KUKA KRL program: EPS_2_251455_MH56A_A_20251003061556.src

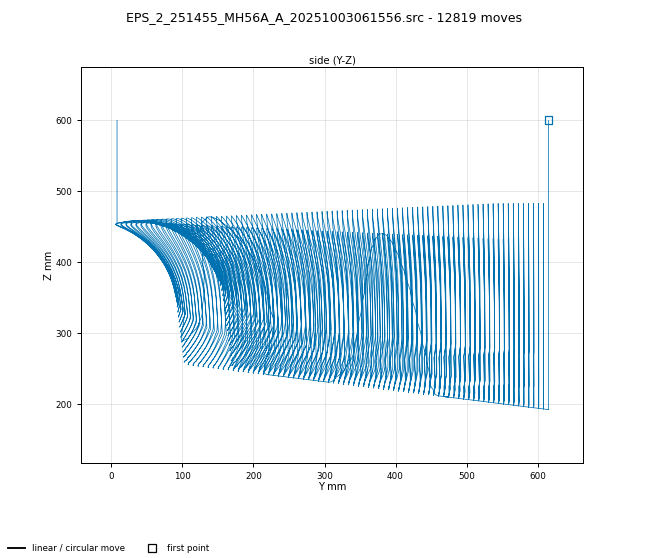
[picture p0: tool path of EPS_2_251455_MH56A_A_20251003061556.src, 12819 of 12821 moves have a stored position in this frame; points joined in program order, loops and branches not executed]
&ACCESS RVP
&REL 4
&COMMENT QRS 19112012
&PARAM EDITMASK = *
DEF PART()
EXT BAS (BAS_COMMAND :IN,REAL :IN )
INT I
BAS (#INITMOV,0 )

;KUKA QRS Post kuka4.cps  Date:22-06-2017 !

File_ID=2879

QRS_PRE_INIT()

;Init var - Until changes are made in qrs_pre_init
Outlet_Square_prg=0
Inlet_1_Square_prg=0
Inlet_2_Square_prg=0
Inlet_3_Square_prg=0
Inlet_4_Square_prg=0
Inlet_5_Square_prg=0

Outlet_1={X 0.000, Y 540.910, Z 382.500, B 0.000, E1 0.000 }
Inlet_1={X 0.000, Y 544.470, Z 332.500, B 0.000, E1 191.000 }
Outlet_1_type=201
Inlet_1_type=201
;QRS#1=Sidecore dimensions
;QRS#2=200-8" PVC SDR 35
;QRS#3=200-8" PVC SDR 35
;QRS#4=
;QRS#5=
;QRS#6=
;QRS#7=
;QRS#8=
;QRS#9=12-08 PSX
;QRS#10=12-08 PSX
;QRS#11=
;QRS#12=
;QRS#13=
;QRS#14=
;QRS#15=
;QRS#16=1220x127x762 2,5'
;QRS#17=EPS Height
;QRS#18=483
;QRS#19=*
;QRS#20= UPDATED VERSION 22-06-2017
;QRS#21=*
Outlet_Square=0100
Inlet_1_Square=0100
Inlet_2_Square=0
Inlet_3_Square=0
Inlet_4_Square=0
Inlet_5_Square=0
Mill_Square=1
Outlet_Square_Prg=204
Inlet_1_Square_prg=204

QRS_INIT()

$ADVANCE=5

; T1
PTP {E1 173.577,E2 173.577}
PTP {X 0,Y 615.465,A -85,B 0,C 180,E1 173.577,E2 173.577,E3 0,E4 0,E5 0,E6 0}
QRS_SPEED_INIT()
LIN {X 0,Y 615.465,Z 600,A -85,B 0,C 180,E1 173.577,E2 173.577,E3 0,E4 0,E5 0,E6 0} C_VEL
LIN {X 0,Y 615.465,Z 202.872,A -85,B 0,C 180,E1 173.577,E2 173.577} C_VEL
LIN {X 0,Y 615.465,Z 194.7,A -85,B 0,C 180,E1 173.577,E2 173.577} C_VEL
LIN {X 0,Y 615.452,Z 192.7,A -85,B 0,C 180,E1 173.391,E2 173.391} C_VEL
LIN {X 0,Y 615.455,Z 192.7,A -85,B 0,C 180,E1 170.801,E2 170.801} C_VEL
LIN {X 0,Y 615.413,Z 192.699,A -85,B 0,C 180,E1 168.138,E2 168.138} C_VEL
LIN {X 0,Y 615.463,Z 192.7,A -85,B 0,C 180,E1 165.45,E2 165.45} C_VEL
LIN {X 0,Y 615.439,Z 192.698,A -85,B 0,C 180,E1 162.728,E2 162.728} C_VEL
LIN {X 0,Y 615.432,Z 192.698,A -85,B 0,C 180,E1 160.66,E2 160.66} C_VEL
LIN {X 0,Y 615.425,Z 192.698,A -85,B 0,C 180,E1 158.566,E2 158.566} C_VEL
LIN {X 0,Y 615.42,Z 192.698,A -85,B 0,C 180,E1 156.441,E2 156.441} C_VEL
LIN {X 0,Y 615.42,Z 192.698,A -85,B 0,C 180,E1 154.281,E2 154.281} C_VEL
LIN {X 0,Y 615.482,Z 192.701,A -85,B 0,C 180,E1 151.538,E2 151.538} C_VEL
LIN {X 0,Y 615.445,Z 192.696,A -85,B 0,C 180,E1 148.909,E2 148.909} C_VEL
LIN {X 0,Y 615.423,Z 192.697,A -85,B 0,C 180,E1 146.464,E2 146.464} C_VEL
LIN {X 0,Y 615.435,Z 192.698,A -85,B 0,C 180,E1 144.163,E2 144.163} C_VEL
LIN {X 0,Y 615.459,Z 192.699,A -85,B 0,C 180,E1 141.929,E2 141.929} C_VEL
LIN {X 0,Y 615.488,Z 192.693,A -85,B 0,C 180,E1 139.393,E2 139.393} C_VEL
LIN {X 0,Y 615.431,Z 192.695,A -85,B 0,C 180,E1 136.75,E2 136.75} C_VEL
LIN {X 0,Y 615.467,Z 192.699,A -85,B 0,C 180,E1 133.995,E2 133.995} C_VEL
LIN {X 0,Y 615.448,Z 192.693,A -85,B 0,C 180,E1 131.09,E2 131.09} C_VEL
LIN {X 0,Y 615.434,Z 192.695,A -85,B 0,C 180,E1 128.902,E2 128.902} C_VEL
LIN {X 0,Y 615.444,Z 192.697,A -85,B 0,C 180,E1 126.422,E2 126.422} C_VEL
LIN {X 0,Y 615.485,Z 192.69,A -85,B 0,C 180,E1 123.533,E2 123.533} C_VEL
LIN {X 0,Y 615.438,Z 192.694,A -85,B 0,C 180,E1 120.918,E2 120.918} C_VEL
LIN {X 0,Y 615.454,Z 192.697,A -85,B 0,C 180,E1 118.444,E2 118.444} C_VEL
LIN {X 0,Y 615.48,Z 192.689,A -85,B 0,C 180,E1 115.566,E2 115.566} C_VEL
LIN {X 0,Y 615.476,Z 192.689,A -85,B 0,C 180,E1 113.553,E2 113.553} C_VEL
LIN {X 0,Y 615.459,Z 192.69,A -85,B 0,C 180,E1 111.429,E2 111.429} C_VEL
LIN {X 0,Y 615.454,Z 192.691,A -85,B 0,C 180,E1 109.336,E2 109.336} C_VEL
LIN {X 0,Y 615.449,Z 192.691,A -85,B 0,C 180,E1 107.269,E2 107.269} C_VEL
LIN {X 0,Y 615.448,Z 192.692,A -85,B 0,C 180,E1 105.224,E2 105.224} C_VEL
LIN {X 0,Y 615.445,Z 192.692,A -85,B 0,C 180,E1 103.2,E2 103.2} C_VEL
LIN {X 0,Y 615.479,Z 192.698,A -85,B 0,C 180,E1 100.525,E2 100.525} C_VEL
LIN {X 0,Y 615.485,Z 192.688,A -85,B 0,C 180,E1 97.874,E2 97.874} C_VEL
LIN {X 0,Y 615.452,Z 192.79,A -85,B 0,C 180,E1 96.973,E2 96.973} C_VEL
LIN {X 0,Y 615.487,Z 208.3,A -85,B 0,C 180,E1 94.255,E2 94.255} C_VEL
LIN {X 0,Y 615.493,Z 222.362,A -85,B 0,C 180,E1 91.818,E2 91.818} C_VEL
LIN {X 0,Y 615.459,Z 329.633,A -85,B 0,C 180,E1 90.53,E2 90.53} C_VEL
LIN {X 0,Y 615.475,Z 342.412,A -85,B 0,C 180,E1 90.244,E2 90.244} C_VEL
LIN {X 0,Y 615.497,Z 354.793,A -85,B 0,C 180,E1 89.835,E2 89.835} C_VEL
LIN {X 0,Y 615.468,Z 365.91,A -85,B 0,C 180,E1 89.345,E2 89.345} C_VEL
LIN {X 0,Y 615.467,Z 377.404,A -85,B 0,C 180,E1 88.69,E2 88.69} C_VEL
LIN {X 0,Y 615.498,Z 388.761,A -85,B 0,C 180,E1 87.872,E2 87.872} C_VEL
LIN {X 0,Y 615.498,Z 397.906,A -85,B 0,C 180,E1 87.054,E2 87.054} C_VEL
LIN {X 0,Y 615.496,Z 406.784,A -85,B 0,C 180,E1 86.071,E2 86.071} C_VEL
LIN {X 0,Y 615.496,Z 413.964,A -85,B 0,C 180,E1 85.087,E2 85.087} C_VEL
LIN {X 0,Y 615.499,Z 419.723,A -85,B 0,C 180,E1 84.101,E2 84.101} C_VEL
LIN {X 0,Y 615.495,Z 424.321,A -85,B 0,C 180,E1 83.101,E2 83.101} C_VEL
LIN {X 0,Y 615.497,Z 427.731,A -85,B 0,C 180,E1 82.124,E2 82.124} C_VEL
LIN {X 0,Y 615.495,Z 429.484,A -85,B 0,C 180,E1 81.463,E2 81.463} C_VEL
LIN {X 0,Y 615.499,Z 431.728,A -85,B 0,C 180,E1 80.138,E2 80.138} C_VEL
LIN {X 0,Y 615.495,Z 432.357,A -85,B 0,C 180,E1 79.11,E2 79.11} C_VEL
LIN {X 0,Y 615.494,Z 432.06,A -85,B 0,C 180,E1 78.139,E2 78.139} C_VEL
LIN {X 0,Y 615.496,Z 431.373,A -85,B 0,C 180,E1 77.47,E2 77.47} C_VEL
LIN {X 0,Y 615.496,Z 430.246,A -85,B 0,C 180,E1 76.799,E2 76.799} C_VEL
LIN {X 0,Y 615.499,Z 428.503,A -85,B 0,C 180,E1 76.065,E2 76.065} C_VEL
LIN {X 0,Y 615.497,Z 425.464,A -85,B 0,C 180,E1 75.113,E2 75.113} C_VEL
LIN {X 0,Y 615.496,Z 421.132,A -85,B 0,C 180,E1 74.095,E2 74.095} C_VEL
LIN {X 0,Y 615.498,Z 415.52,A -85,B 0,C 180,E1 73.072,E2 73.072} C_VEL
LIN {X 0,Y 615.499,Z 408.424,A -85,B 0,C 180,E1 72.044,E2 72.044} C_VEL
LIN {X 0,Y 615.497,Z 401.088,A -85,B 0,C 180,E1 71.182,E2 71.182} C_VEL
LIN {X 0,Y 615.498,Z 391.05,A -85,B 0,C 180,E1 70.229,E2 70.229} C_VEL
LIN {X 0,Y 615.489,Z 380.813,A -85,B 0,C 180,E1 69.444,E2 69.444} C_VEL
LIN {X 0,Y 615.462,Z 369.296,A -85,B 0,C 180,E1 68.744,E2 68.744} C_VEL
LIN {X 0,Y 615.491,Z 357.249,A -85,B 0,C 180,E1 68.173,E2 68.173} C_VEL
LIN {X 0,Y 615.446,Z 345.875,A -85,B 0,C 180,E1 67.764,E2 67.764} C_VEL
LIN {X 0,Y 615.433,Z 333.072,A -85,B 0,C 180,E1 67.442,E2 67.442} C_VEL
LIN {X 0,Y 615.436,Z 317.595,A -85,B 0,C 180,E1 67.218,E2 67.218} C_VEL
LIN {X 0,Y 615.479,Z 222.383,A -85,B 0,C 180,E1 66.095,E2 66.095} C_VEL
LIN {X 0,Y 615.491,Z 206.009,A -85,B 0,C 180,E1 63.257,E2 63.257} C_VEL
LIN {X 0,Y 615.469,Z 192.69,A -85,B 0,C 180,E1 60.899,E2 60.899} C_VEL
LIN {X 0,Y 615.489,Z 192.684,A -85,B 0,C 180,E1 58.317,E2 58.317} C_VEL
LIN {X 0,Y 615.483,Z 192.692,A -85,B 0,C 180,E1 55.98,E2 55.98} C_VEL
LIN {X 0,Y 615.484,Z 192.701,A -85,B 0,C 180,E1 53.578,E2 53.578} C_VEL
LIN {X 0,Y 615.462,Z 192.689,A -85,B 0,C 180,E1 50.941,E2 50.941} C_VEL
LIN {X 0,Y 615.489,Z 192.683,A -85,B 0,C 180,E1 48.53,E2 48.53} C_VEL
LIN {X 0,Y 615.498,Z 192.699,A -85,B 0,C 180,E1 45.855,E2 45.855} C_VEL
LIN {X 0,Y 615.46,Z 192.689,A -85,B 0,C 180,E1 43.049,E2 43.049} C_VEL
LIN {X 0,Y 615.49,Z 192.684,A -85,B 0,C 180,E1 40.607,E2 40.607} C_VEL
LIN {X 0,Y 615.484,Z 192.703,A -85,B 0,C 180,E1 38.017,E2 38.017} C_VEL
LIN {X 0,Y 615.461,Z 192.696,A -85,B 0,C 180,E1 35.618,E2 35.618} C_VEL
LIN {X 0,Y 615.452,Z 192.691,A -85,B 0,C 180,E1 33.239,E2 33.239} C_VEL
LIN {X 0,Y 615.471,Z 192.687,A -85,B 0,C 180,E1 30.921,E2 30.921} C_VEL
LIN {X 0,Y 615.469,Z 192.697,A -85,B 0,C 180,E1 27.916,E2 27.916} C_VEL
LIN {X 0,Y 615.445,Z 192.694,A -85,B 0,C 180,E1 25.569,E2 25.569} C_VEL
LIN {X 0,Y 615.487,Z 192.687,A -85,B 0,C 180,E1 22.845,E2 22.845} C_VEL
LIN {X 0,Y 615.462,Z 192.697,A -85,B 0,C 180,E1 20.034,E2 20.034} C_VEL
LIN {X 0,Y 615.453,Z 192.697,A -85,B 0,C 180,E1 17.958,E2 17.958} C_VEL
LIN {X 0,Y 615.446,Z 192.696,A -85,B 0,C 180,E1 15.906,E2 15.906} C_VEL
LIN {X 0,Y 615.442,Z 192.696,A -85,B 0,C 180,E1 13.875,E2 13.875} C_VEL
LIN {X 0,Y 615.439,Z 192.696,A -85,B 0,C 180,E1 11.862,E2 11.862} C_VEL
LIN {X 0,Y 615.437,Z 192.696,A -85,B 0,C 180,E1 9.863,E2 9.863} C_VEL
LIN {X 0,Y 615.434,Z 192.696,A -85,B 0,C 180,E1 7.876,E2 7.876} C_VEL
LIN {X 0,Y 615.461,Z 192.693,A -85,B 0,C 180,E1 5.242,E2 5.242} C_VEL
LIN {X 0,Y 615.478,Z 192.701,A -85,B 0,C 180,E1 2.618,E2 2.618} C_VEL
LIN {X 0,Y 615.429,Z 192.697,A -85,B 0,C 180,E1 0,E2 0} C_VEL
LIN {X 0,Y 615.454,Z 192.695,A -85,B 0,C 180,E1 -2.618,E2 -2.618} C_VEL
LIN {X 0,Y 615.475,Z 192.7,A -85,B 0,C 180,E1 -5.241,E2 -5.241} C_VEL
LIN {X 0,Y 615.42,Z 192.699,A -85,B 0,C 180,E1 -7.876,E2 -7.876} C_VEL
LIN {X 0,Y 615.451,Z 192.697,A -85,B 0,C 180,E1 -10.528,E2 -10.528} C_VEL
LIN {X 0,Y 615.457,Z 192.7,A -85,B 0,C 180,E1 -13.202,E2 -13.202} C_VEL
LIN {X 0,Y 615.414,Z 192.699,A -85,B 0,C 180,E1 -15.907,E2 -15.907} C_VEL
LIN {X 0,Y 615.469,Z 192.701,A -85,B 0,C 180,E1 -18.647,E2 -18.647} C_VEL
LIN {X 0,Y 615.419,Z 192.7,A -85,B 0,C 180,E1 -21.434,E2 -21.434} C_VEL
LIN {X 0,Y 615.415,Z 192.7,A -85,B 0,C 180,E1 -23.559,E2 -23.559} C_VEL
LIN {X 0,Y 615.414,Z 192.699,A -85,B 0,C 180,E1 -25.719,E2 -25.719} C_VEL
LIN {X 0,Y 615.473,Z 192.701,A -85,B 0,C 180,E1 -28.456,E2 -28.456} C_VEL
LIN {X 0,Y 615.443,Z 192.697,A -85,B 0,C 180,E1 -31.086,E2 -31.086} C_VEL
LIN {X 0,Y 615.42,Z 192.698,A -85,B 0,C 180,E1 -33.531,E2 -33.531} C_VEL
LIN {X 0,Y 615.431,Z 192.698,A -85,B 0,C 180,E1 -35.832,E2 -35.832} C_VEL
LIN {X 0,Y 615.456,Z 192.699,A -85,B 0,C 180,E1 -38.071,E2 -38.071} C_VEL
LIN {X 0,Y 615.485,Z 192.694,A -85,B 0,C 180,E1 -40.607,E2 -40.607} C_VEL
LIN {X 0,Y 615.431,Z 192.695,A -85,B 0,C 180,E1 -43.25,E2 -43.25} C_VEL
LIN {X 0,Y 615.467,Z 192.699,A -85,B 0,C 180,E1 -46.005,E2 -46.005} C_VEL
LIN {X 0,Y 615.449,Z 192.693,A -85,B 0,C 180,E1 -48.91,E2 -48.91} C_VEL
LIN {X 0,Y 615.436,Z 192.694,A -85,B 0,C 180,E1 -51.095,E2 -51.095} C_VEL
LIN {X 0,Y 615.446,Z 192.697,A -85,B 0,C 180,E1 -53.575,E2 -53.575} C_VEL
LIN {X 0,Y 615.486,Z 192.689,A -85,B 0,C 180,E1 -56.466,E2 -56.466} C_VEL
LIN {X 0,Y 615.442,Z 192.693,A -85,B 0,C 180,E1 -59.08,E2 -59.08} C_VEL
LIN {X 0,Y 615.458,Z 192.698,A -85,B 0,C 180,E1 -61.555,E2 -61.555} C_VEL
LIN {X 0,Y 615.48,Z 192.688,A -85,B 0,C 180,E1 -64.433,E2 -64.433} C_VEL
LIN {X 0,Y 615.447,Z 192.693,A -85,B 0,C 180,E1 -67.044,E2 -67.044} C_VEL
LIN {X 0,Y 615.482,Z 210.777,A -85,B 0,C 180,E1 -69.445,E2 -69.445} C_VEL
LIN {X 0,Y 615.489,Z 232.021,A -85,B 0,C 180,E1 -72.215,E2 -72.215} C_VEL
LIN {X 0,Y 615.494,Z 253.241,A -85,B 0,C 180,E1 -74.944,E2 -74.944} C_VEL
LIN {X 0,Y 615.452,Z 270.301,A -85,B 0,C 180,E1 -77.113,E2 -77.113} C_VEL
LIN {X 0,Y 615.478,Z 378.826,A -85,B 0,C 180,E1 -78.41,E2 -78.41} C_VEL
LIN {X 0,Y 615.47,Z 391.342,A -85,B 0,C 180,E1 -78.681,E2 -78.681} C_VEL
LIN {X 0,Y 615.486,Z 404.641,A -85,B 0,C 180,E1 -79.114,E2 -79.114} C_VEL
LIN {X 0,Y 615.483,Z 416.473,A -85,B 0,C 180,E1 -79.639,E2 -79.639} C_VEL
LIN {X 0,Y 615.495,Z 427.989,A -85,B 0,C 180,E1 -80.304,E2 -80.304} C_VEL
LIN {X 0,Y 615.499,Z 438.336,A -85,B 0,C 180,E1 -81.049,E2 -81.049} C_VEL
LIN {X 0,Y 615.497,Z 446.807,A -85,B 0,C 180,E1 -81.794,E2 -81.794} C_VEL
LIN {X 0,Y 615.498,Z 454.602,A -85,B 0,C 180,E1 -82.619,E2 -82.619} C_VEL
LIN {X 0,Y 615.496,Z 462.199,A -85,B 0,C 180,E1 -83.607,E2 -83.607} C_VEL
LIN {X 0,Y 615.498,Z 469.201,A -85,B 0,C 180,E1 -84.758,E2 -84.758} C_VEL
LIN {X 0,Y 615.494,Z 473.848,A -85,B 0,C 180,E1 -85.743,E2 -85.743} C_VEL
LIN {X 0,Y 615.494,Z 477.396,A -85,B 0,C 180,E1 -86.726,E2 -86.726} C_VEL
LIN {X 0,Y 615.497,Z 479.23,A -85,B 0,C 180,E1 -87.381,E2 -87.381} C_VEL
LIN {X 0,Y 615.499,Z 480.606,A -85,B 0,C 180,E1 -88.036,E2 -88.036} C_VEL
LIN {X 0,Y 615.496,Z 482.173,A -85,B 0,C 180,E1 -89.345,E2 -89.345} C_VEL
LIN {X 0,Y 615.494,Z 482.389,A -85,B 0,C 180,E1 -89.999,E2 -89.999} C_VEL
LIN {X 0,Y 615.495,Z 481.582,A -85,B 0,C 180,E1 -91.307,E2 -91.307} C_VEL
LIN {X 0,Y 615.499,Z 480.61,A -85,B 0,C 180,E1 -91.962,E2 -91.962} C_VEL
LIN {X 0,Y 615.497,Z 479.237,A -85,B 0,C 180,E1 -92.616,E2 -92.616} C_VEL
LIN {X 0,Y 615.496,Z 476.355,A -85,B 0,C 180,E1 -93.599,E2 -93.599} C_VEL
LIN {X 0,Y 615.498,Z 472.449,A -85,B 0,C 180,E1 -94.583,E2 -94.583} C_VEL
LIN {X 0,Y 615.499,Z 467.415,A -85,B 0,C 180,E1 -95.568,E2 -95.568} C_VEL
LIN {X 0,Y 615.496,Z 460.87,A -85,B 0,C 180,E1 -96.583,E2 -96.583} C_VEL
LIN {X 0,Y 615.497,Z 453.151,A -85,B 0,C 180,E1 -97.543,E2 -97.543} C_VEL
LIN {X 0,Y 615.498,Z 445.067,A -85,B 0,C 180,E1 -98.369,E2 -98.369} C_VEL
LIN {X 0,Y 615.499,Z 435.196,A -85,B 0,C 180,E1 -99.196,E2 -99.196} C_VEL
LIN {X 0,Y 615.492,Z 424.018,A -85,B 0,C 180,E1 -99.943,E2 -99.943} C_VEL
LIN {X 0,Y 615.485,Z 413.071,A -85,B 0,C 180,E1 -100.525,E2 -100.525} C_VEL
LIN {X 0,Y 615.476,Z 400.537,A -85,B 0,C 180,E1 -101.039,E2 -101.039} C_VEL
LIN {X 0,Y 615.471,Z 388.173,A -85,B 0,C 180,E1 -101.399,E2 -101.399} C_VEL
LIN {X 0,Y 615.481,Z 374.641,A -85,B 0,C 180,E1 -101.65,E2 -101.65} C_VEL
LIN {X 0,Y 615.452,Z 270.321,A -85,B 0,C 180,E1 -102.885,E2 -102.885} C_VEL
LIN {X 0,Y 615.487,Z 249.282,A -85,B 0,C 180,E1 -105.562,E2 -105.562} C_VEL
LIN {X 0,Y 615.456,Z 227.019,A -85,B 0,C 180,E1 -108.434,E2 -108.434} C_VEL
LIN {X 0,Y 615.482,Z 206.808,A -85,B 0,C 180,E1 -111.078,E2 -111.078} C_VEL
LIN {X 0,Y 615.447,Z 192.693,A -85,B 0,C 180,E1 -112.976,E2 -112.976} C_VEL
LIN {X 0,Y 615.499,Z 192.686,A -85,B 0,C 180,E1 -115.711,E2 -115.711} C_VEL
LIN {X 0,Y 615.45,Z 192.695,A -85,B 0,C 180,E1 -118.655,E2 -118.655} C_VEL
LIN {X 0,Y 615.447,Z 192.692,A -85,B 0,C 180,E1 -121.079,E2 -121.079} C_VEL
LIN {X 0,Y 615.495,Z 192.701,A -85,B 0,C 180,E1 -124.016,E2 -124.016} C_VEL
LIN {X 0,Y 615.454,Z 192.697,A -85,B 0,C 180,E1 -126.421,E2 -126.421} C_VEL
LIN {X 0,Y 615.445,Z 192.692,A -85,B 0,C 180,E1 -129.057,E2 -129.057} C_VEL
LIN {X 0,Y 615.487,Z 192.689,A -85,B 0,C 180,E1 -131.467,E2 -131.467} C_VEL
LIN {X 0,Y 615.464,Z 192.698,A -85,B 0,C 180,E1 -134.145,E2 -134.145} C_VEL
LIN {X 0,Y 615.437,Z 192.694,A -85,B 0,C 180,E1 -136.751,E2 -136.751} C_VEL
LIN {X 0,Y 615.489,Z 192.691,A -85,B 0,C 180,E1 -139.394,E2 -139.394} C_VEL
LIN {X 0,Y 615.465,Z 192.699,A -85,B 0,C 180,E1 -141.982,E2 -141.982} C_VEL
LIN {X 0,Y 615.433,Z 192.696,A -85,B 0,C 180,E1 -144.38,E2 -144.38} C_VEL
LIN {X 0,Y 615.436,Z 192.694,A -85,B 0,C 180,E1 -146.761,E2 -146.761} C_VEL
LIN {X 0,Y 615.465,Z 192.693,A -85,B 0,C 180,E1 -149.079,E2 -149.079} C_VEL
LIN {X 0,Y 615.439,Z 192.698,A -85,B 0,C 180,E1 -152.082,E2 -152.082} C_VEL
LIN {X 0,Y 615.427,Z 192.696,A -85,B 0,C 180,E1 -154.428,E2 -154.428} C_VEL
LIN {X 0,Y 615.484,Z 192.694,A -85,B 0,C 180,E1 -157.155,E2 -157.155} C_VEL
LIN {X 0,Y 615.435,Z 192.698,A -85,B 0,C 180,E1 -159.965,E2 -159.965} C_VEL
LIN {X 0,Y 615.429,Z 192.698,A -85,B 0,C 180,E1 -162.041,E2 -162.041} C_VEL
LIN {X 0,Y 615.425,Z 192.698,A -85,B 0,C 180,E1 -164.093,E2 -164.093} C_VEL
LIN {X 0,Y 615.422,Z 192.698,A -85,B 0,C 180,E1 -166.124,E2 -166.124} C_VEL
LIN {X 0,Y 615.455,Z 192.696,A -85,B 0,C 180,E1 -168.806,E2 -168.806} C_VEL
LIN {X 0,Y 615.461,Z 192.7,A -85,B 0,C 180,E1 -171.463,E2 -171.463} C_VEL
LIN {X 0,Y 615.417,Z 192.699,A -85,B 0,C 180,E1 -174.101,E2 -174.101} C_VEL
LIN {X 0,Y 615.455,Z 192.698,A -85,B 0,C 180,E1 -176.727,E2 -176.727} C_VEL
LIN {X 0,Y 615.457,Z 192.7,A -85,B 0,C 180,E1 -179.346,E2 -179.346} C_VEL
LIN {X 0,Y 615.413,Z 192.7,A -85,B 0,C 180,E1 -181.963,E2 -181.963} C_VEL
LIN {X 0,Y 615.447,Z 192.7,A -85,B 0,C 180,E1 -184.585,E2 -184.585} C_VEL
LIN {X 0,Y 615.452,Z 192.7,A -85,B 0,C 180,E1 -186.609,E2 -186.609} C_VEL
LIN {X 0,Y 614.78,Z 192.847,A -85,B 0,C 180,E1 -187.155,E2 -187.155} C_VEL
LIN {X 0,Y 611.949,Z 193.252,A -85,B 0,C 180,E1 -188.041,E2 -188.041} C_VEL
LIN {X 0,Y 609.552,Z 193.564,A -85,B 0,C 180,E1 -188.753,E2 -188.753} C_VEL
LIN {X 0,Y 608.505,Z 193.685,A -85,B 0,C 180,E1 -189.303,E2 -189.303} C_VEL
LIN {X 0,Y 608.409,Z 193.694,A -85,B 0,C 180,E1 -189.489,E2 -189.489} C_VEL
LIN {X 0,Y 608.427,Z 193.694,A -85,B 0,C 180,E1 -191.325,E2 -191.325} C_VEL
LIN {X 0,Y 608.403,Z 193.694,A -85,B 0,C 180,E1 -194.039,E2 -194.039} C_VEL
LIN {X 0,Y 608.439,Z 193.699,A -85,B 0,C 180,E1 -196.785,E2 -196.785} C_VEL
LIN {X 0,Y 608.395,Z 193.695,A -85,B 0,C 180,E1 -199.573,E2 -199.573} C_VEL
LIN {X 0,Y 608.411,Z 193.692,A -85,B 0,C 180,E1 -201.694,E2 -201.694} C_VEL
LIN {X 0,Y 608.418,Z 193.702,A -85,B 0,C 180,E1 -204.573,E2 -204.573} C_VEL
LIN {X 0,Y 608.398,Z 193.694,A -85,B 0,C 180,E1 -207.521,E2 -207.521} C_VEL
LIN {X 0,Y 608.416,Z 193.694,A -85,B 0,C 180,E1 -209.975,E2 -209.975} C_VEL
LIN {X 0,Y 608.456,Z 193.697,A -85,B 0,C 180,E1 -212.533,E2 -212.533} C_VEL
LIN {X 0,Y 608.4,Z 193.694,A -85,B 0,C 180,E1 -215.281,E2 -215.281} C_VEL
LIN {X 0,Y 608.429,Z 193.692,A -85,B 0,C 180,E1 -217.749,E2 -217.749} C_VEL
LIN {X 0,Y 608.441,Z 193.7,A -85,B 0,C 180,E1 -220.336,E2 -220.336} C_VEL
LIN {X 0,Y 608.414,Z 193.693,A -85,B 0,C 180,E1 -222.964,E2 -222.964} C_VEL
LIN {X 0,Y 608.41,Z 193.693,A -85,B 0,C 180,E1 -225.207,E2 -225.207} C_VEL
LIN {X 0,Y 608.441,Z 193.695,A -85,B 0,C 180,E1 -227.944,E2 -227.944} C_VEL
LIN {X 0,Y 608.446,Z 193.69,A -85,B 0,C 180,E1 -230.706,E2 -230.706} C_VEL
LIN {X 0,Y 608.409,Z 193.693,A -85,B 0,C 180,E1 -233.088,E2 -233.088} C_VEL
LIN {X 0,Y 608.436,Z 193.692,A -85,B 0,C 180,E1 -235.534,E2 -235.534} C_VEL
LIN {X 0,Y 608.448,Z 193.697,A -85,B 0,C 180,E1 -237.909,E2 -237.909} C_VEL
LIN {X 0,Y 608.479,Z 193.691,A -85,B 0,C 180,E1 -240.226,E2 -240.226} C_VEL
LIN {X 0,Y 608.409,Z 193.694,A -85,B 0,C 180,E1 -243.228,E2 -243.228} C_VEL
LIN {X 0,Y 608.481,Z 193.694,A -85,B 0,C 180,E1 -245.848,E2 -245.848} C_VEL
LIN {X 0,Y 608.455,Z 193.69,A -85,B 0,C 180,E1 -248.312,E2 -248.312} C_VEL
LIN {X 0,Y 608.434,Z 193.691,A -85,B 0,C 180,E1 -251.133,E2 -251.133} C_VEL
LIN {X 0,Y 608.46,Z 193.694,A -85,B 0,C 180,E1 -253.909,E2 -253.909} C_VEL
LIN {X 0,Y 608.437,Z 193.689,A -85,B 0,C 180,E1 -256.646,E2 -256.646} C_VEL
LIN {X 0,Y 608.448,Z 193.693,A -85,B 0,C 180,E1 -259.352,E2 -259.352} C_VEL
LIN {X 0,Y 608.476,Z 193.688,A -85,B 0,C 180,E1 -262.035,E2 -262.035} C_VEL
LIN {X 0,Y 608.458,Z 193.89,A -85,B 0,C 180,E1 -262.994,E2 -262.994} C_VEL
LIN {X 0,Y 608.471,Z 209.187,A -85,B 0,C 180,E1 -265.696,E2 -265.696} C_VEL
LIN {X 0,Y 608.472,Z 222.602,A -85,B 0,C 180,E1 -268.036,E2 -268.036} C_VEL
LIN {X 0,Y 608.523,Z 328.822,A -85,B 0,C 180,E1 -269.319,E2 -269.319} C_VEL
LIN {X 0,Y 608.527,Z 341.914,A -85,B 0,C 180,E1 -269.608,E2 -269.608} C_VEL
LIN {X 0,Y 608.527,Z 355.032,A -85,B 0,C 180,E1 -270.043,E2 -270.043} C_VEL
LIN {X 0,Y 608.49,Z 366.942,A -85,B 0,C 180,E1 -270.58,E2 -270.58} C_VEL
LIN {X 0,Y 608.456,Z 378.296,A -85,B 0,C 180,E1 -271.242,E2 -271.242} C_VEL
LIN {X 0,Y 608.472,Z 388.545,A -85,B 0,C 180,E1 -271.987,E2 -271.987} C_VEL
LIN {X 0,Y 608.477,Z 397.847,A -85,B 0,C 180,E1 -272.815,E2 -272.815} C_VEL
LIN {X 0,Y 608.458,Z 406.848,A -85,B 0,C 180,E1 -273.809,E2 -273.809} C_VEL
LIN {X 0,Y 608.463,Z 414.136,A -85,B 0,C 180,E1 -274.804,E2 -274.804} C_VEL
LIN {X 0,Y 608.438,Z 420.843,A -85,B 0,C 180,E1 -275.968,E2 -275.968} C_VEL
LIN {X 0,Y 608.442,Z 425.288,A -85,B 0,C 180,E1 -276.967,E2 -276.967} C_VEL
LIN {X 0,Y 608.424,Z 428.666,A -85,B 0,C 180,E1 -277.968,E2 -277.968} C_VEL
LIN {X 0,Y 608.42,Z 430.343,A -85,B 0,C 180,E1 -278.637,E2 -278.637} C_VEL
LIN {X 0,Y 608.421,Z 431.613,A -85,B 0,C 180,E1 -279.307,E2 -279.307} C_VEL
LIN {X 0,Y 608.434,Z 432.484,A -85,B 0,C 180,E1 -279.978,E2 -279.978} C_VEL
LIN {X 0,Y 608.422,Z 432.979,A -85,B 0,C 180,E1 -280.931,E2 -280.931} C_VEL
LIN {X 0,Y 608.439,Z 432.577,A -85,B 0,C 180,E1 -282,E2 -282} C_VEL
LIN {X 0,Y 608.42,Z 431.787,A -85,B 0,C 180,E1 -282.678,E2 -282.678} C_VEL
LIN {X 0,Y 608.439,Z 430.551,A -85,B 0,C 180,E1 -283.357,E2 -283.357} C_VEL
LIN {X 0,Y 608.428,Z 427.88,A -85,B 0,C 180,E1 -284.38,E2 -284.38} C_VEL
LIN {X 0,Y 608.426,Z 424.132,A -85,B 0,C 180,E1 -285.407,E2 -285.407} C_VEL
LIN {X 0,Y 608.433,Z 418.754,A -85,B 0,C 180,E1 -286.517,E2 -286.517} C_VEL
LIN {X 0,Y 608.452,Z 412.855,A -85,B 0,C 180,E1 -287.476,E2 -287.476} C_VEL
LIN {X 0,Y 608.474,Z 405.06,A -85,B 0,C 180,E1 -288.499,E2 -288.499} C_VEL
LIN {X 0,Y 608.486,Z 396.61,A -85,B 0,C 180,E1 -289.393,E2 -289.393} C_VEL
LIN {X 0,Y 608.478,Z 386.399,A -85,B 0,C 180,E1 -290.273,E2 -290.273} C_VEL
LIN {X 0,Y 608.464,Z 376.265,A -85,B 0,C 180,E1 -290.98,E2 -290.98} C_VEL
LIN {X 0,Y 608.483,Z 365.113,A -85,B 0,C 180,E1 -291.601,E2 -291.601} C_VEL
LIN {X 0,Y 608.511,Z 352.713,A -85,B 0,C 180,E1 -292.135,E2 -292.135} C_VEL
LIN {X 0,Y 608.503,Z 339.502,A -85,B 0,C 180,E1 -292.548,E2 -292.548} C_VEL
LIN {X 0,Y 608.494,Z 326.057,A -85,B 0,C 180,E1 -292.812,E2 -292.812} C_VEL
LIN {X 0,Y 608.452,Z 222.74,A -85,B 0,C 180,E1 -294.043,E2 -294.043} C_VEL
LIN {X 0,Y 608.457,Z 208.087,A -85,B 0,C 180,E1 -296.587,E2 -296.587} C_VEL
LIN {X 0,Y 608.453,Z 193.689,A -85,B 0,C 180,E1 -299.161,E2 -299.161} C_VEL
LIN {X 0,Y 608.472,Z 193.69,A -85,B 0,C 180,E1 -302.092,E2 -302.092} C_VEL
LIN {X 0,Y 608.463,Z 193.689,A -85,B 0,C 180,E1 -304.907,E2 -304.907} C_VEL
LIN {X 0,Y 608.466,Z 193.688,A -85,B 0,C 180,E1 -307.744,E2 -307.744} C_VEL
LIN {X 0,Y 608.47,Z 193.695,A -85,B 0,C 180,E1 -310.331,E2 -310.331} C_VEL
LIN {X 0,Y 608.433,Z 193.691,A -85,B 0,C 180,E1 -312.958,E2 -312.958} C_VEL
LIN {X 0,Y 608.454,Z 193.691,A -85,B 0,C 180,E1 -315.732,E2 -315.732} C_VEL
LIN {X 0,Y 608.436,Z 193.692,A -85,B 0,C 180,E1 -318.656,E2 -318.656} C_VEL
LIN {X 0,Y 608.455,Z 193.689,A -85,B 0,C 180,E1 -321.411,E2 -321.411} C_VEL
LIN {X 0,Y 608.46,Z 193.697,A -85,B 0,C 180,E1 -323.947,E2 -323.947} C_VEL
LIN {X 0,Y 608.444,Z 193.692,A -85,B 0,C 180,E1 -326.328,E2 -326.328} C_VEL
LIN {X 0,Y 608.449,Z 193.688,A -85,B 0,C 180,E1 -328.725,E2 -328.725} C_VEL
LIN {X 0,Y 608.472,Z 193.688,A -85,B 0,C 180,E1 -331.373,E2 -331.373} C_VEL
LIN {X 0,Y 608.433,Z 193.692,A -85,B 0,C 180,E1 -334.278,E2 -334.278} C_VEL
LIN {X 0,Y 608.432,Z 193.69,A -85,B 0,C 180,E1 -336.875,E2 -336.875} C_VEL
LIN {X 0,Y 608.452,Z 193.697,A -85,B 0,C 180,E1 -339.725,E2 -339.725} C_VEL
LIN {X 0,Y 608.429,Z 193.697,A -85,B 0,C 180,E1 -341.827,E2 -341.827} C_VEL
LIN {X 0,Y 608.435,Z 193.694,A -85,B 0,C 180,E1 -343.905,E2 -343.905} C_VEL
LIN {X 0,Y 608.433,Z 193.693,A -85,B 0,C 180,E1 -345.979,E2 -345.979} C_VEL
LIN {X 0,Y 608.443,Z 193.689,A -85,B 0,C 180,E1 -348.676,E2 -348.676} C_VEL
LIN {X 0,Y 608.449,Z 193.698,A -85,B 0,C 180,E1 -351.364,E2 -351.364} C_VEL
LIN {X 0,Y 608.412,Z 193.693,A -85,B 0,C 180,E1 -354.033,E2 -354.033} C_VEL
LIN {X 0,Y 608.45,Z 193.69,A -85,B 0,C 180,E1 -356.689,E2 -356.689} C_VEL
LIN {X 0,Y 608.472,Z 193.694,A -85,B 0,C 180,E1 -359.338,E2 -359.338} C_VEL
LIN {X 0,Y 608.398,Z 193.695,A -85,B 0,C 180,E1 -361.986,E2 -361.986} C_VEL
LIN {X 0,Y 608.396,Z 193.695,A -85,B 0,C 180,E1 -363.974,E2 -363.974} C_VEL
LIN {X 0,Y 608.434,Z 193.693,A -85,B 0,C 180,E1 -366.633,E2 -366.633} C_VEL
LIN {X 0,Y 608.444,Z 193.694,A -85,B 0,C 180,E1 -369.306,E2 -369.306} C_VEL
LIN {X 0,Y 608.443,Z 193.693,A -85,B 0,C 180,E1 -371.324,E2 -371.324} C_VEL
LIN {X 0,Y 608.403,Z 193.694,A -85,B 0,C 180,E1 -374.039,E2 -374.039} C_VEL
LIN {X 0,Y 608.443,Z 193.698,A -85,B 0,C 180,E1 -376.784,E2 -376.784} C_VEL
LIN {X 0,Y 608.393,Z 193.695,A -85,B 0,C 180,E1 -379.573,E2 -379.573} C_VEL
LIN {X 0,Y 608.405,Z 193.693,A -85,B 0,C 180,E1 -381.694,E2 -381.694} C_VEL
LIN {X 0,Y 608.423,Z 193.693,A -85,B 0,C 180,E1 -384.15,E2 -384.15} C_VEL
LIN {X 0,Y 608.421,Z 193.7,A -85,B 0,C 180,E1 -386.776,E2 -386.776} C_VEL
LIN {X 0,Y 608.435,Z 193.693,A -85,B 0,C 180,E1 -389.022,E2 -389.022} C_VEL
LIN {X 0,Y 608.407,Z 193.694,A -85,B 0,C 180,E1 -391.32,E2 -391.32} C_VEL
LIN {X 0,Y 608.394,Z 193.695,A -85,B 0,C 180,E1 -393.73,E2 -393.73} C_VEL
LIN {X 0,Y 608.418,Z 193.696,A -85,B 0,C 180,E1 -396.094,E2 -396.094} C_VEL
LIN {X 0,Y 608.439,Z 193.696,A -85,B 0,C 180,E1 -398.59,E2 -398.59} C_VEL
LIN {X 0,Y 608.402,Z 193.694,A -85,B 0,C 180,E1 -401.181,E2 -401.181} C_VEL
LIN {X 0,Y 608.424,Z 193.691,A -85,B 0,C 180,E1 -403.308,E2 -403.308} C_VEL
LIN {X 0,Y 608.452,Z 193.697,A -85,B 0,C 180,E1 -406.133,E2 -406.133} C_VEL
LIN {X 0,Y 608.426,Z 193.692,A -85,B 0,C 180,E1 -408.824,E2 -408.824} C_VEL
LIN {X 0,Y 608.448,Z 193.693,A -85,B 0,C 180,E1 -411.762,E2 -411.762} C_VEL
LIN {X 0,Y 608.431,Z 193.691,A -85,B 0,C 180,E1 -414.724,E2 -414.724} C_VEL
LIN {X 0,Y 608.43,Z 193.69,A -85,B 0,C 180,E1 -417.121,E2 -417.121} C_VEL
LIN {X 0,Y 608.473,Z 193.694,A -85,B 0,C 180,E1 -420.028,E2 -420.028} C_VEL
LIN {X 0,Y 608.449,Z 193.688,A -85,B 0,C 180,E1 -422.799,E2 -422.799} C_VEL
LIN {X 0,Y 608.437,Z 193.694,A -85,B 0,C 180,E1 -425.429,E2 -425.429} C_VEL
LIN {X 0,Y 608.449,Z 193.828,A -85,B 0,C 180,E1 -426.922,E2 -426.922} C_VEL
LIN {X 0,Y 608.58,Z 209.449,A -85,B 0,C 180,E1 -429.024,E2 -429.024} C_VEL
LIN {X 0,Y 608.522,Z 230.721,A -85,B 0,C 180,E1 -431.831,E2 -431.831} C_VEL
LIN {X 0,Y 608.489,Z 251.992,A -85,B 0,C 180,E1 -434.595,E2 -434.595} C_VEL
LIN {X 0,Y 608.45,Z 270.522,A -85,B 0,C 180,E1 -436.973,E2 -436.973} C_VEL
LIN {X 0,Y 608.539,Z 378.941,A -85,B 0,C 180,E1 -438.276,E2 -438.276} C_VEL
LIN {X 0,Y 608.505,Z 392.211,A -85,B 0,C 180,E1 -438.571,E2 -438.571} C_VEL
LIN {X 0,Y 608.513,Z 404.638,A -85,B 0,C 180,E1 -438.983,E2 -438.983} C_VEL
LIN {X 0,Y 608.504,Z 416.63,A -85,B 0,C 180,E1 -439.519,E2 -439.519} C_VEL
LIN {X 0,Y 608.486,Z 428.193,A -85,B 0,C 180,E1 -440.191,E2 -440.191} C_VEL
LIN {X 0,Y 608.485,Z 438.589,A -85,B 0,C 180,E1 -440.945,E2 -440.945} C_VEL
LIN {X 0,Y 608.475,Z 447.107,A -85,B 0,C 180,E1 -441.698,E2 -441.698} C_VEL
LIN {X 0,Y 608.471,Z 454.956,A -85,B 0,C 180,E1 -442.533,E2 -442.533} C_VEL
LIN {X 0,Y 608.461,Z 462.284,A -85,B 0,C 180,E1 -443.484,E2 -443.484} C_VEL
LIN {X 0,Y 608.45,Z 467.862,A -85,B 0,C 180,E1 -444.365,E2 -444.365} C_VEL
LIN {X 0,Y 608.432,Z 472.947,A -85,B 0,C 180,E1 -445.361,E2 -445.361} C_VEL
LIN {X 0,Y 608.449,Z 476.893,A -85,B 0,C 180,E1 -446.357,E2 -446.357} C_VEL
LIN {X 0,Y 608.425,Z 479.807,A -85,B 0,C 180,E1 -447.351,E2 -447.351} C_VEL
LIN {X 0,Y 608.444,Z 481.2,A -85,B 0,C 180,E1 -448.013,E2 -448.013} C_VEL
LIN {X 0,Y 608.439,Z 482.783,A -85,B 0,C 180,E1 -449.337,E2 -449.337} C_VEL
LIN {X 0,Y 608.434,Z 483,A -85,B 0,C 180,E1 -449.999,E2 -449.999} C_VEL
LIN {X 0,Y 608.448,Z 482.185,A -85,B 0,C 180,E1 -451.322,E2 -451.322} C_VEL
LIN {X 0,Y 608.444,Z 481.204,A -85,B 0,C 180,E1 -451.984,E2 -451.984} C_VEL
LIN {X 0,Y 608.425,Z 479.813,A -85,B 0,C 180,E1 -452.647,E2 -452.647} C_VEL
LIN {X 0,Y 608.449,Z 476.901,A -85,B 0,C 180,E1 -453.641,E2 -453.641} C_VEL
LIN {X 0,Y 608.432,Z 472.957,A -85,B 0,C 180,E1 -454.636,E2 -454.636} C_VEL
LIN {X 0,Y 608.437,Z 466.888,A -85,B 0,C 180,E1 -455.799,E2 -455.799} C_VEL
LIN {X 0,Y 608.461,Z 460.249,A -85,B 0,C 180,E1 -456.797,E2 -456.797} C_VEL
LIN {X 0,Y 608.455,Z 452.007,A -85,B 0,C 180,E1 -457.798,E2 -457.798} C_VEL
LIN {X 0,Y 608.471,Z 443.56,A -85,B 0,C 180,E1 -458.634,E2 -458.634} C_VEL
LIN {X 0,Y 608.479,Z 433.121,A -85,B 0,C 180,E1 -459.471,E2 -459.471} C_VEL
LIN {X 0,Y 608.496,Z 422.794,A -85,B 0,C 180,E1 -460.142,E2 -460.142} C_VEL
LIN {X 0,Y 608.519,Z 411.309,A -85,B 0,C 180,E1 -460.738,E2 -460.738} C_VEL
LIN {X 0,Y 608.523,Z 398.953,A -85,B 0,C 180,E1 -461.223,E2 -461.223} C_VEL
LIN {X 0,Y 608.535,Z 385.543,A -85,B 0,C 180,E1 -461.595,E2 -461.595} C_VEL
LIN {X 0,Y 608.547,Z 373.268,A -85,B 0,C 180,E1 -461.805,E2 -461.805} C_VEL
LIN {X 0,Y 608.438,Z 270.459,A -85,B 0,C 180,E1 -463.036,E2 -463.036} C_VEL
LIN {X 0,Y 608.5,Z 249.353,A -85,B 0,C 180,E1 -465.746,E2 -465.746} C_VEL
LIN {X 0,Y 608.5,Z 228.273,A -85,B 0,C 180,E1 -468.491,E2 -468.491} C_VEL
LIN {X 0,Y 608.556,Z 208.139,A -85,B 0,C 180,E1 -471.152,E2 -471.152} C_VEL
LIN {X 0,Y 608.446,Z 193.765,A -85,B 0,C 180,E1 -473.087,E2 -473.087} C_VEL
LIN {X 0,Y 608.474,Z 193.688,A -85,B 0,C 180,E1 -475.721,E2 -475.721} C_VEL
LIN {X 0,Y 608.446,Z 193.691,A -85,B 0,C 180,E1 -478.615,E2 -478.615} C_VEL
LIN {X 0,Y 608.449,Z 193.691,A -85,B 0,C 180,E1 -480.541,E2 -480.541} C_VEL
LIN {X 0,Y 608.43,Z 193.69,A -85,B 0,C 180,E1 -482.876,E2 -482.876} C_VEL
LIN {X 0,Y 608.43,Z 193.691,A -85,B 0,C 180,E1 -485.273,E2 -485.273} C_VEL
LIN {X 0,Y 608.451,Z 193.693,A -85,B 0,C 180,E1 -488.238,E2 -488.238} C_VEL
LIN {X 0,Y 608.426,Z 193.695,A -85,B 0,C 180,E1 -490.326,E2 -490.326} C_VEL
LIN {X 0,Y 608.416,Z 193.692,A -85,B 0,C 180,E1 -492.956,E2 -492.956} C_VEL
LIN {X 0,Y 608.454,Z 193.696,A -85,B 0,C 180,E1 -495.729,E2 -495.729} C_VEL
LIN {X 0,Y 608.458,Z 193.695,A -85,B 0,C 180,E1 -497.938,E2 -497.938} C_VEL
LIN {X 0,Y 608.433,Z 193.69,A -85,B 0,C 180,E1 -500.698,E2 -500.698} C_VEL
LIN {X 0,Y 608.429,Z 193.692,A -85,B 0,C 180,E1 -503.083,E2 -503.083} C_VEL
LIN {X 0,Y 608.455,Z 193.696,A -85,B 0,C 180,E1 -505.53,E2 -505.53} C_VEL
LIN {X 0,Y 608.448,Z 193.693,A -85,B 0,C 180,E1 -507.904,E2 -507.904} C_VEL
LIN {X 0,Y 608.42,Z 193.693,A -85,B 0,C 180,E1 -510.218,E2 -510.218} C_VEL
LIN {X 0,Y 608.436,Z 193.69,A -85,B 0,C 180,E1 -512.787,E2 -512.787} C_VEL
LIN {X 0,Y 608.437,Z 193.694,A -85,B 0,C 180,E1 -515.841,E2 -515.841} C_VEL
LIN {X 0,Y 608.418,Z 193.692,A -85,B 0,C 180,E1 -518.307,E2 -518.307} C_VEL
LIN {X 0,Y 608.4,Z 193.694,A -85,B 0,C 180,E1 -520.428,E2 -520.428} C_VEL
LIN {X 0,Y 608.466,Z 193.694,A -85,B 0,C 180,E1 -523.448,E2 -523.448} C_VEL
LIN {X 0,Y 608.408,Z 193.694,A -85,B 0,C 180,E1 -525.979,E2 -525.979} C_VEL
LIN {X 0,Y 608.405,Z 193.694,A -85,B 0,C 180,E1 -527.999,E2 -527.999} C_VEL
LIN {X 0,Y 608.397,Z 193.695,A -85,B 0,C 180,E1 -530.022,E2 -530.022} C_VEL
LIN {X 0,Y 608.438,Z 193.692,A -85,B 0,C 180,E1 -532.7,E2 -532.7} C_VEL
LIN {X 0,Y 608.426,Z 193.697,A -85,B 0,C 180,E1 -535.362,E2 -535.362} C_VEL
LIN {X 0,Y 608.386,Z 193.696,A -85,B 0,C 180,E1 -538.014,E2 -538.014} C_VEL
LIN {X 0,Y 608.442,Z 193.693,A -85,B 0,C 180,E1 -540.662,E2 -540.662} C_VEL
LIN {X 0,Y 608.444,Z 193.693,A -85,B 0,C 180,E1 -543.311,E2 -543.311} C_VEL
LIN {X 0,Y 608.388,Z 193.695,A -85,B 0,C 180,E1 -545.968,E2 -545.968} C_VEL
LIN {X 0,Y 608.416,Z 193.698,A -85,B 0,C 180,E1 -548.637,E2 -548.637} C_VEL
LIN {X 0,Y 608.409,Z 193.694,A -85,B 0,C 180,E1 -549.489,E2 -549.489} C_VEL
LIN {X 0,Y 607.712,Z 193.782,A -85,B 0,C 180,E1 -550.042,E2 -550.042} C_VEL
LIN {X 0,Y 604.84,Z 194.147,A -85,B 0,C 180,E1 -550.939,E2 -550.939} C_VEL
LIN {X 0,Y 602.445,Z 194.44,A -85,B 0,C 180,E1 -551.661,E2 -551.661} C_VEL
LIN {X 0,Y 601.439,Z 194.563,A -85,B 0,C 180,E1 -552.218,E2 -552.218} C_VEL
LIN {X 0,Y 601.368,Z 194.573,A -85,B 0,C 180,E1 -552.406,E2 -552.406} C_VEL
LIN {X 0,Y 601.388,Z 194.576,A -85,B 0,C 180,E1 -554.898,E2 -554.898} C_VEL
LIN {X 0,Y 601.386,Z 194.574,A -85,B 0,C 180,E1 -556.987,E2 -556.987} C_VEL
LIN {X 0,Y 601.355,Z 194.572,A -85,B 0,C 180,E1 -559.811,E2 -559.811} C_VEL
LIN {X 0,Y 601.371,Z 194.571,A -85,B 0,C 180,E1 -561.961,E2 -561.961} C_VEL
LIN {X 0,Y 601.387,Z 194.573,A -85,B 0,C 180,E1 -564.298,E2 -564.298} C_VEL
LIN {X 0,Y 601.409,Z 194.567,A -85,B 0,C 180,E1 -567.113,E2 -567.113} C_VEL
LIN {X 0,Y 601.372,Z 194.57,A -85,B 0,C 180,E1 -569.396,E2 -569.396} C_VEL
LIN {X 0,Y 601.374,Z 194.57,A -85,B 0,C 180,E1 -571.729,E2 -571.729} C_VEL
LIN {X 0,Y 601.392,Z 194.572,A -85,B 0,C 180,E1 -574.121,E2 -574.121} C_VEL
LIN {X 0,Y 601.377,Z 194.576,A -85,B 0,C 180,E1 -576.585,E2 -576.585} C_VEL
LIN {X 0,Y 601.371,Z 194.57,A -85,B 0,C 180,E1 -579.13,E2 -579.13} C_VEL
LIN {X 0,Y 601.391,Z 194.569,A -85,B 0,C 180,E1 -581.768,E2 -581.768} C_VEL
LIN {X 0,Y 601.388,Z 194.573,A -85,B 0,C 180,E1 -584.539,E2 -584.539} C_VEL
LIN {X 0,Y 601.373,Z 194.569,A -85,B 0,C 180,E1 -587.333,E2 -587.333} C_VEL
LIN {X 0,Y 601.384,Z 194.576,A -85,B 0,C 180,E1 -590.009,E2 -590.009} C_VEL
LIN {X 0,Y 601.409,Z 194.568,A -85,B 0,C 180,E1 -592.622,E2 -592.622} C_VEL
LIN {X 0,Y 601.373,Z 194.569,A -85,B 0,C 180,E1 -595.071,E2 -595.071} C_VEL
LIN {X 0,Y 601.396,Z 194.569,A -85,B 0,C 180,E1 -597.487,E2 -597.487} C_VEL
LIN {X 0,Y 601.433,Z 194.57,A -85,B 0,C 180,E1 -599.851,E2 -599.851} C_VEL
LIN {X 0,Y 601.397,Z 194.566,A -85,B 0,C 180,E1 -602.891,E2 -602.891} C_VEL
LIN {X 0,Y 601.433,Z 194.569,A -85,B 0,C 180,E1 -605.709,E2 -605.709} C_VEL
LIN {X 0,Y 601.398,Z 194.573,A -85,B 0,C 180,E1 -608.044,E2 -608.044} C_VEL
LIN {X 0,Y 601.402,Z 194.566,A -85,B 0,C 180,E1 -610.904,E2 -610.904} C_VEL
LIN {X 0,Y 601.424,Z 194.573,A -85,B 0,C 180,E1 -613.716,E2 -613.716} C_VEL
LIN {X 0,Y 601.399,Z 194.566,A -85,B 0,C 180,E1 -616.486,E2 -616.486} C_VEL
LIN {X 0,Y 601.389,Z 194.571,A -85,B 0,C 180,E1 -619.226,E2 -619.226} C_VEL
LIN {X 0,Y 601.439,Z 194.567,A -85,B 0,C 180,E1 -621.941,E2 -621.941} C_VEL
LIN {X 0,Y 601.4,Z 194.648,A -85,B 0,C 180,E1 -622.912,E2 -622.912} C_VEL
LIN {X 0,Y 601.44,Z 206.16,A -85,B 0,C 180,E1 -624.974,E2 -624.974} C_VEL
LIN {X 0,Y 601.418,Z 222.64,A -85,B 0,C 180,E1 -627.888,E2 -627.888} C_VEL
LIN {X 0,Y 601.68,Z 237.632,A -85,B 0,C 180,E1 -628.077,E2 -628.077} C_VEL
LIN {X 0,Y 601.584,Z 329.03,A -85,B 0,C 180,E1 -629.186,E2 -629.186} C_VEL
LIN {X 0,Y 601.577,Z 342.054,A -85,B 0,C 180,E1 -629.478,E2 -629.478} C_VEL
LIN {X 0,Y 601.553,Z 355.143,A -85,B 0,C 180,E1 -629.918,E2 -629.918} C_VEL
LIN {X 0,Y 601.509,Z 366.227,A -85,B 0,C 180,E1 -630.42,E2 -630.42} C_VEL
LIN {X 0,Y 601.435,Z 377.737,A -85,B 0,C 180,E1 -631.089,E2 -631.089} C_VEL
LIN {X 0,Y 601.465,Z 388.074,A -85,B 0,C 180,E1 -631.842,E2 -631.842} C_VEL
LIN {X 0,Y 601.41,Z 397.474,A -85,B 0,C 180,E1 -632.68,E2 -632.68} C_VEL
LIN {X 0,Y 601.376,Z 406.55,A -85,B 0,C 180,E1 -633.686,E2 -633.686} C_VEL
LIN {X 0,Y 601.401,Z 413.885,A -85,B 0,C 180,E1 -634.693,E2 -634.693} C_VEL
LIN {X 0,Y 601.373,Z 419.795,A -85,B 0,C 180,E1 -635.702,E2 -635.702} C_VEL
LIN {X 0,Y 601.36,Z 424.471,A -85,B 0,C 180,E1 -636.712,E2 -636.712} C_VEL
LIN {X 0,Y 601.338,Z 428.05,A -85,B 0,C 180,E1 -637.725,E2 -637.725} C_VEL
LIN {X 0,Y 601.332,Z 430.624,A -85,B 0,C 180,E1 -638.74,E2 -638.74} C_VEL
LIN {X 0,Y 601.336,Z 431.828,A -85,B 0,C 180,E1 -639.418,E2 -639.418} C_VEL
LIN {X 0,Y 601.329,Z 432.591,A -85,B 0,C 180,E1 -640.097,E2 -640.097} C_VEL
LIN {X 0,Y 601.336,Z 432.988,A -85,B 0,C 180,E1 -640.966,E2 -640.966} C_VEL
LIN {X 0,Y 601.342,Z 432.464,A -85,B 0,C 180,E1 -642.144,E2 -642.144} C_VEL
LIN {X 0,Y 601.326,Z 431.57,A -85,B 0,C 180,E1 -642.83,E2 -642.83} C_VEL
LIN {X 0,Y 601.352,Z 428.916,A -85,B 0,C 180,E1 -644.064,E2 -644.064} C_VEL
LIN {X 0,Y 601.354,Z 425.014,A -85,B 0,C 180,E1 -645.245,E2 -645.245} C_VEL
LIN {X 0,Y 601.356,Z 420.324,A -85,B 0,C 180,E1 -646.289,E2 -646.289} C_VEL
LIN {X 0,Y 601.395,Z 414.285,A -85,B 0,C 180,E1 -647.337,E2 -647.337} C_VEL
LIN {X 0,Y 601.375,Z 406.64,A -85,B 0,C 180,E1 -648.393,E2 -648.393} C_VEL
LIN {X 0,Y 601.417,Z 398.784,A -85,B 0,C 180,E1 -649.276,E2 -649.276} C_VEL
LIN {X 0,Y 601.457,Z 389.13,A -85,B 0,C 180,E1 -650.163,E2 -650.163} C_VEL
LIN {X 0,Y 601.45,Z 378.472,A -85,B 0,C 180,E1 -650.952,E2 -650.952} C_VEL
LIN {X 0,Y 601.501,Z 367.65,A -85,B 0,C 180,E1 -651.594,E2 -651.594} C_VEL
LIN {X 0,Y 601.527,Z 355.153,A -85,B 0,C 180,E1 -652.173,E2 -652.173} C_VEL
LIN {X 0,Y 601.526,Z 342.321,A -85,B 0,C 180,E1 -652.605,E2 -652.605} C_VEL
LIN {X 0,Y 601.551,Z 329.125,A -85,B 0,C 180,E1 -652.903,E2 -652.903} C_VEL
LIN {X 0,Y 601.572,Z 223.941,A -85,B 0,C 180,E1 -654.18,E2 -654.18} C_VEL
LIN {X 0,Y 601.382,Z 222.589,A -85,B 0,C 180,E1 -654.212,E2 -654.212} C_VEL
LIN {X 0,Y 601.437,Z 208.303,A -85,B 0,C 180,E1 -656.735,E2 -656.735} C_VEL
LIN {X 0,Y 601.449,Z 194.563,A -85,B 0,C 180,E1 -659.222,E2 -659.222} C_VEL
LIN {X 0,Y 601.401,Z 194.567,A -85,B 0,C 180,E1 -661.725,E2 -661.725} C_VEL
LIN {X 0,Y 601.424,Z 194.569,A -85,B 0,C 180,E1 -664.116,E2 -664.116} C_VEL
LIN {X 0,Y 601.399,Z 194.573,A -85,B 0,C 180,E1 -666.581,E2 -666.581} C_VEL
LIN {X 0,Y 601.431,Z 194.563,A -85,B 0,C 180,E1 -669.534,E2 -669.534} C_VEL
LIN {X 0,Y 601.422,Z 194.567,A -85,B 0,C 180,E1 -671.762,E2 -671.762} C_VEL
LIN {X 0,Y 601.408,Z 194.57,A -85,B 0,C 180,E1 -674.533,E2 -674.533} C_VEL
LIN {X 0,Y 601.424,Z 194.564,A -85,B 0,C 180,E1 -677.404,E2 -677.404} C_VEL
LIN {X 0,Y 601.422,Z 194.567,A -85,B 0,C 180,E1 -680.462,E2 -680.462} C_VEL
LIN {X 0,Y 601.413,Z 194.566,A -85,B 0,C 180,E1 -682.616,E2 -682.616} C_VEL
LIN {X 0,Y 601.419,Z 194.564,A -85,B 0,C 180,E1 -685.068,E2 -685.068} C_VEL
LIN {X 0,Y 601.429,Z 194.566,A -85,B 0,C 180,E1 -687.484,E2 -687.484} C_VEL
LIN {X 0,Y 601.423,Z 194.574,A -85,B 0,C 180,E1 -689.845,E2 -689.845} C_VEL
LIN {X 0,Y 601.405,Z 194.57,A -85,B 0,C 180,E1 -692.132,E2 -692.132} C_VEL
LIN {X 0,Y 601.381,Z 194.57,A -85,B 0,C 180,E1 -695.12,E2 -695.12} C_VEL
LIN {X 0,Y 601.427,Z 194.568,A -85,B 0,C 180,E1 -697.382,E2 -697.382} C_VEL
LIN {X 0,Y 601.38,Z 194.57,A -85,B 0,C 180,E1 -700.19,E2 -700.19} C_VEL
LIN {X 0,Y 601.407,Z 194.567,A -85,B 0,C 180,E1 -703.013,E2 -703.013} C_VEL
LIN {X 0,Y 601.384,Z 194.572,A -85,B 0,C 180,E1 -705.905,E2 -705.905} C_VEL
LIN {X 0,Y 601.399,Z 194.566,A -85,B 0,C 180,E1 -708.541,E2 -708.541} C_VEL
LIN {X 0,Y 601.423,Z 194.571,A -85,B 0,C 180,E1 -711.262,E2 -711.262} C_VEL
LIN {X 0,Y 601.37,Z 194.571,A -85,B 0,C 180,E1 -713.962,E2 -713.962} C_VEL
LIN {X 0,Y 601.4,Z 194.568,A -85,B 0,C 180,E1 -716.65,E2 -716.65} C_VEL
LIN {X 0,Y 601.439,Z 194.57,A -85,B 0,C 180,E1 -719.33,E2 -719.33} C_VEL
LIN {X 0,Y 601.37,Z 194.57,A -85,B 0,C 180,E1 -722.009,E2 -722.009} C_VEL
LIN {X 0,Y 601.35,Z 194.572,A -85,B 0,C 180,E1 -724.021,E2 -724.021} C_VEL
LIN {X 0,Y 601.411,Z 194.569,A -85,B 0,C 180,E1 -726.711,E2 -726.711} C_VEL
LIN {X 0,Y 601.385,Z 194.572,A -85,B 0,C 180,E1 -729.416,E2 -729.416} C_VEL
LIN {X 0,Y 601.395,Z 194.569,A -85,B 0,C 180,E1 -731.459,E2 -731.459} C_VEL
LIN {X 0,Y 601.371,Z 194.571,A -85,B 0,C 180,E1 -734.207,E2 -734.207} C_VEL
LIN {X 0,Y 601.393,Z 194.575,A -85,B 0,C 180,E1 -736.987,E2 -736.987} C_VEL
LIN {X 0,Y 601.353,Z 194.572,A -85,B 0,C 180,E1 -739.811,E2 -739.811} C_VEL
LIN {X 0,Y 601.362,Z 194.571,A -85,B 0,C 180,E1 -741.961,E2 -741.961} C_VEL
LIN {X 0,Y 601.386,Z 194.572,A -85,B 0,C 180,E1 -744.291,E2 -744.291} C_VEL
LIN {X 0,Y 601.36,Z 194.572,A -85,B 0,C 180,E1 -747.36,E2 -747.36} C_VEL
LIN {X 0,Y 601.373,Z 194.57,A -85,B 0,C 180,E1 -749.396,E2 -749.396} C_VEL
LIN {X 0,Y 601.368,Z 194.57,A -85,B 0,C 180,E1 -751.729,E2 -751.729} C_VEL
LIN {X 0,Y 601.388,Z 194.572,A -85,B 0,C 180,E1 -754.121,E2 -754.121} C_VEL
LIN {X 0,Y 601.374,Z 194.577,A -85,B 0,C 180,E1 -756.585,E2 -756.585} C_VEL
LIN {X 0,Y 601.374,Z 194.569,A -85,B 0,C 180,E1 -759.13,E2 -759.13} C_VEL
LIN {X 0,Y 601.395,Z 194.569,A -85,B 0,C 180,E1 -761.768,E2 -761.768} C_VEL
LIN {X 0,Y 601.406,Z 194.571,A -85,B 0,C 180,E1 -764.537,E2 -764.537} C_VEL
LIN {X 0,Y 601.36,Z 194.571,A -85,B 0,C 180,E1 -767.329,E2 -767.329} C_VEL
LIN {X 0,Y 601.388,Z 194.576,A -85,B 0,C 180,E1 -770.006,E2 -770.006} C_VEL
LIN {X 0,Y 601.419,Z 194.566,A -85,B 0,C 180,E1 -772.62,E2 -772.62} C_VEL
LIN {X 0,Y 601.377,Z 194.569,A -85,B 0,C 180,E1 -775.068,E2 -775.068} C_VEL
LIN {X 0,Y 601.403,Z 194.568,A -85,B 0,C 180,E1 -777.485,E2 -777.485} C_VEL
LIN {X 0,Y 601.424,Z 194.572,A -85,B 0,C 180,E1 -779.853,E2 -779.853} C_VEL
LIN {X 0,Y 601.404,Z 194.566,A -85,B 0,C 180,E1 -782.888,E2 -782.888} C_VEL
LIN {X 0,Y 601.461,Z 194.569,A -85,B 0,C 180,E1 -785.861,E2 -785.861} C_VEL
LIN {X 0,Y 601.406,Z 194.658,A -85,B 0,C 180,E1 -786.75,E2 -786.75} C_VEL
LIN {X 0,Y 601.696,Z 199.704,A -85,B 0,C 180,E1 -787.451,E2 -787.451} C_VEL
LIN {X 0,Y 601.598,Z 220.085,A -85,B 0,C 180,E1 -790.198,E2 -790.198} C_VEL
LIN {X 0,Y 601.529,Z 241.356,A -85,B 0,C 180,E1 -793.017,E2 -793.017} C_VEL
LIN {X 0,Y 601.458,Z 262.628,A -85,B 0,C 180,E1 -795.796,E2 -795.796} C_VEL
LIN {X 0,Y 601.425,Z 270.522,A -85,B 0,C 180,E1 -796.818,E2 -796.818} C_VEL
LIN {X 0,Y 601.617,Z 287.24,A -85,B 0,C 180,E1 -797.026,E2 -797.026} C_VEL
LIN {X 0,Y 601.606,Z 378.941,A -85,B 0,C 180,E1 -798.139,E2 -798.139} C_VEL
LIN {X 0,Y 601.569,Z 392.212,A -85,B 0,C 180,E1 -798.438,E2 -798.438} C_VEL
LIN {X 0,Y 601.542,Z 404.638,A -85,B 0,C 180,E1 -798.853,E2 -798.853} C_VEL
LIN {X 0,Y 601.525,Z 416.629,A -85,B 0,C 180,E1 -799.396,E2 -799.396} C_VEL
LIN {X 0,Y 601.486,Z 428.194,A -85,B 0,C 180,E1 -800.076,E2 -800.076} C_VEL
LIN {X 0,Y 601.444,Z 438.591,A -85,B 0,C 180,E1 -800.839,E2 -800.839} C_VEL
LIN {X 0,Y 601.429,Z 447.107,A -85,B 0,C 180,E1 -801.6,E2 -801.6} C_VEL
LIN {X 0,Y 601.418,Z 454.956,A -85,B 0,C 180,E1 -802.445,E2 -802.445} C_VEL
LIN {X 0,Y 601.37,Z 462.222,A -85,B 0,C 180,E1 -803.398,E2 -803.398} C_VEL
LIN {X 0,Y 601.372,Z 467.862,A -85,B 0,C 180,E1 -804.298,E2 -804.298} C_VEL
LIN {X 0,Y 601.336,Z 472.947,A -85,B 0,C 180,E1 -805.307,E2 -805.307} C_VEL
LIN {X 0,Y 601.368,Z 476.893,A -85,B 0,C 180,E1 -806.314,E2 -806.314} C_VEL
LIN {X 0,Y 601.325,Z 479.806,A -85,B 0,C 180,E1 -807.319,E2 -807.319} C_VEL
LIN {X 0,Y 601.343,Z 481.2,A -85,B 0,C 180,E1 -807.99,E2 -807.99} C_VEL
LIN {X 0,Y 601.339,Z 482.783,A -85,B 0,C 180,E1 -809.329,E2 -809.329} C_VEL
LIN {X 0,Y 601.335,Z 483,A -85,B 0,C 180,E1 -809.999,E2 -809.999} C_VEL
LIN {X 0,Y 601.347,Z 482.186,A -85,B 0,C 180,E1 -811.338,E2 -811.338} C_VEL
LIN {X 0,Y 601.343,Z 481.204,A -85,B 0,C 180,E1 -812.008,E2 -812.008} C_VEL
LIN {X 0,Y 601.325,Z 479.813,A -85,B 0,C 180,E1 -812.678,E2 -812.678} C_VEL
LIN {X 0,Y 601.368,Z 476.901,A -85,B 0,C 180,E1 -813.684,E2 -813.684} C_VEL
LIN {X 0,Y 601.336,Z 472.957,A -85,B 0,C 180,E1 -814.691,E2 -814.691} C_VEL
LIN {X 0,Y 601.372,Z 466.888,A -85,B 0,C 180,E1 -815.867,E2 -815.867} C_VEL
LIN {X 0,Y 601.386,Z 460.25,A -85,B 0,C 180,E1 -816.878,E2 -816.878} C_VEL
LIN {X 0,Y 601.4,Z 452.007,A -85,B 0,C 180,E1 -817.89,E2 -817.89} C_VEL
LIN {X 0,Y 601.436,Z 443.561,A -85,B 0,C 180,E1 -818.735,E2 -818.735} C_VEL
LIN {X 0,Y 601.449,Z 433.123,A -85,B 0,C 180,E1 -819.583,E2 -819.583} C_VEL
LIN {X 0,Y 601.473,Z 422.796,A -85,B 0,C 180,E1 -820.262,E2 -820.262} C_VEL
LIN {X 0,Y 601.535,Z 410.624,A -85,B 0,C 180,E1 -820.895,E2 -820.895} C_VEL
LIN {X 0,Y 601.549,Z 398.286,A -85,B 0,C 180,E1 -821.377,E2 -821.377} C_VEL
LIN {X 0,Y 601.571,Z 385.542,A -85,B 0,C 180,E1 -821.731,E2 -821.731} C_VEL
LIN {X 0,Y 601.614,Z 373.268,A -85,B 0,C 180,E1 -821.943,E2 -821.943} C_VEL
LIN {X 0,Y 601.535,Z 271.359,A -85,B 0,C 180,E1 -823.167,E2 -823.167} C_VEL
LIN {X 0,Y 601.431,Z 270.459,A -85,B 0,C 180,E1 -823.19,E2 -823.19} C_VEL
LIN {X 0,Y 601.521,Z 248.024,A -85,B 0,C 180,E1 -826.107,E2 -826.107} C_VEL
LIN {X 0,Y 601.585,Z 225.423,A -85,B 0,C 180,E1 -829.09,E2 -829.09} C_VEL
LIN {X 0,Y 601.677,Z 204.151,A -85,B 0,C 180,E1 -831.945,E2 -831.945} C_VEL
LIN {X 0,Y 601.657,Z 196.174,A -85,B 0,C 180,E1 -833.033,E2 -833.033} C_VEL
LIN {X 0,Y 601.392,Z 194.571,A -85,B 0,C 180,E1 -833.271,E2 -833.271} C_VEL
LIN {X 0,Y 601.413,Z 194.57,A -85,B 0,C 180,E1 -835.867,E2 -835.867} C_VEL
LIN {X 0,Y 601.404,Z 194.568,A -85,B 0,C 180,E1 -838.624,E2 -838.624} C_VEL
LIN {X 0,Y 601.393,Z 194.567,A -85,B 0,C 180,E1 -840.939,E2 -840.939} C_VEL
LIN {X 0,Y 601.423,Z 194.572,A -85,B 0,C 180,E1 -843.934,E2 -843.934} C_VEL
LIN {X 0,Y 601.381,Z 194.57,A -85,B 0,C 180,E1 -846.579,E2 -846.579} C_VEL
LIN {X 0,Y 601.42,Z 194.567,A -85,B 0,C 180,E1 -849.533,E2 -849.533} C_VEL
LIN {X 0,Y 601.406,Z 194.574,A -85,B 0,C 180,E1 -851.76,E2 -851.76} C_VEL
LIN {X 0,Y 601.388,Z 194.568,A -85,B 0,C 180,E1 -854.531,E2 -854.531} C_VEL
LIN {X 0,Y 601.421,Z 194.567,A -85,B 0,C 180,E1 -857.4,E2 -857.4} C_VEL
LIN {X 0,Y 601.401,Z 194.567,A -85,B 0,C 180,E1 -860.46,E2 -860.46} C_VEL
LIN {X 0,Y 601.393,Z 194.567,A -85,B 0,C 180,E1 -862.614,E2 -862.614} C_VEL
LIN {X 0,Y 601.408,Z 194.567,A -85,B 0,C 180,E1 -865.067,E2 -865.067} C_VEL
LIN {X 0,Y 601.45,Z 194.568,A -85,B 0,C 180,E1 -867.485,E2 -867.485} C_VEL
LIN {X 0,Y 601.399,Z 194.572,A -85,B 0,C 180,E1 -869.844,E2 -869.844} C_VEL
LIN {X 0,Y 601.387,Z 194.569,A -85,B 0,C 180,E1 -872.131,E2 -872.131} C_VEL
LIN {X 0,Y 601.377,Z 194.569,A -85,B 0,C 180,E1 -874.38,E2 -874.38} C_VEL
LIN {X 0,Y 601.38,Z 194.569,A -85,B 0,C 180,E1 -876.588,E2 -876.588} C_VEL
LIN {X 0,Y 601.412,Z 194.574,A -85,B 0,C 180,E1 -879.477,E2 -879.477} C_VEL
LIN {X 0,Y 601.385,Z 194.574,A -85,B 0,C 180,E1 -881.607,E2 -881.607} C_VEL
LIN {X 0,Y 601.407,Z 194.569,A -85,B 0,C 180,E1 -883.712,E2 -883.712} C_VEL
LIN {X 0,Y 601.368,Z 194.57,A -85,B 0,C 180,E1 -886.483,E2 -886.483} C_VEL
LIN {X 0,Y 601.407,Z 194.576,A -85,B 0,C 180,E1 -889.224,E2 -889.224} C_VEL
LIN {X 0,Y 601.381,Z 194.569,A -85,B 0,C 180,E1 -891.938,E2 -891.938} C_VEL
LIN {X 0,Y 601.352,Z 194.572,A -85,B 0,C 180,E1 -893.962,E2 -893.962} C_VEL
LIN {X 0,Y 601.392,Z 194.57,A -85,B 0,C 180,E1 -896.65,E2 -896.65} C_VEL
LIN {X 0,Y 601.415,Z 194.57,A -85,B 0,C 180,E1 -899.331,E2 -899.331} C_VEL
LIN {X 0,Y 601.355,Z 194.572,A -85,B 0,C 180,E1 -902.009,E2 -902.009} C_VEL
LIN {X 0,Y 601.383,Z 194.574,A -85,B 0,C 180,E1 -904.692,E2 -904.692} C_VEL
LIN {X 0,Y 601.399,Z 194.569,A -85,B 0,C 180,E1 -907.386,E2 -907.386} C_VEL
LIN {X 0,Y 601.373,Z 194.57,A -85,B 0,C 180,E1 -910.096,E2 -910.096} C_VEL
LIN {X 0,Y 601.368,Z 194.573,A -85,B 0,C 180,E1 -912.406,E2 -912.406} C_VEL
LIN {X 0,Y 600.729,Z 194.66,A -85,B 0,C 180,E1 -912.966,E2 -912.966} C_VEL
LIN {X 0,Y 597.878,Z 195.016,A -85,B 0,C 180,E1 -913.873,E2 -913.873} C_VEL
LIN {X 0,Y 595.448,Z 195.316,A -85,B 0,C 180,E1 -914.603,E2 -914.603} C_VEL
LIN {X 0,Y 594.4,Z 195.442,A -85,B 0,C 180,E1 -915.167,E2 -915.167} C_VEL
LIN {X 0,Y 594.314,Z 195.451,A -85,B 0,C 180,E1 -915.358,E2 -915.358} C_VEL
LIN {X 0,Y 594.328,Z 195.447,A -85,B 0,C 180,E1 -917.906,E2 -917.906} C_VEL
LIN {X 0,Y 594.379,Z 195.449,A -85,B 0,C 180,E1 -920.777,E2 -920.777} C_VEL
LIN {X 0,Y 594.342,Z 195.445,A -85,B 0,C 180,E1 -923.706,E2 -923.706} C_VEL
LIN {X 0,Y 594.344,Z 195.453,A -85,B 0,C 180,E1 -926.702,E2 -926.702} C_VEL
LIN {X 0,Y 594.372,Z 195.445,A -85,B 0,C 180,E1 -928.999,E2 -928.999} C_VEL
LIN {X 0,Y 594.347,Z 195.445,A -85,B 0,C 180,E1 -931.649,E2 -931.649} C_VEL
LIN {X 0,Y 594.36,Z 195.451,A -85,B 0,C 180,E1 -934.582,E2 -934.582} C_VEL
LIN {X 0,Y 594.344,Z 195.446,A -85,B 0,C 180,E1 -937.09,E2 -937.09} C_VEL
LIN {X 0,Y 594.324,Z 195.449,A -85,B 0,C 180,E1 -939.777,E2 -939.777} C_VEL
LIN {X 0,Y 594.363,Z 195.452,A -85,B 0,C 180,E1 -942.376,E2 -942.376} C_VEL
LIN {X 0,Y 594.328,Z 195.447,A -85,B 0,C 180,E1 -945.195,E2 -945.195} C_VEL
LIN {X 0,Y 594.334,Z 195.448,A -85,B 0,C 180,E1 -947.628,E2 -947.628} C_VEL
LIN {X 0,Y 594.368,Z 195.45,A -85,B 0,C 180,E1 -950.325,E2 -950.325} C_VEL
LIN {X 0,Y 594.356,Z 195.444,A -85,B 0,C 180,E1 -952.917,E2 -952.917} C_VEL
LIN {X 0,Y 594.361,Z 195.45,A -85,B 0,C 180,E1 -955.865,E2 -955.865} C_VEL
LIN {X 0,Y 594.35,Z 195.446,A -85,B 0,C 180,E1 -958.653,E2 -958.653} C_VEL
LIN {X 0,Y 594.36,Z 195.443,A -85,B 0,C 180,E1 -961.047,E2 -961.047} C_VEL
LIN {X 0,Y 594.38,Z 195.45,A -85,B 0,C 180,E1 -963.979,E2 -963.979} C_VEL
LIN {X 0,Y 594.371,Z 195.445,A -85,B 0,C 180,E1 -966.299,E2 -966.299} C_VEL
LIN {X 0,Y 594.38,Z 195.442,A -85,B 0,C 180,E1 -969.227,E2 -969.227} C_VEL
LIN {X 0,Y 594.34,Z 195.45,A -85,B 0,C 180,E1 -972.098,E2 -972.098} C_VEL
LIN {X 0,Y 594.351,Z 195.447,A -85,B 0,C 180,E1 -974.222,E2 -974.222} C_VEL
LIN {X 0,Y 594.369,Z 195.443,A -85,B 0,C 180,E1 -976.323,E2 -976.323} C_VEL
LIN {X 0,Y 594.349,Z 195.447,A -85,B 0,C 180,E1 -979.097,E2 -979.097} C_VEL
LIN {X 0,Y 594.411,Z 195.445,A -85,B 0,C 180,E1 -981.845,E2 -981.845} C_VEL
LIN {X 0,Y 594.395,Z 195.635,A -85,B 0,C 180,E1 -982.87,E2 -982.87} C_VEL
LIN {X 0,Y 594.42,Z 206.912,A -85,B 0,C 180,E1 -984.914,E2 -984.914} C_VEL
LIN {X 0,Y 594.384,Z 222.557,A -85,B 0,C 180,E1 -987.714,E2 -987.714} C_VEL
LIN {X 0,Y 594.74,Z 227.551,A -85,B 0,C 180,E1 -987.801,E2 -987.801} C_VEL
LIN {X 0,Y 594.637,Z 329.247,A -85,B 0,C 180,E1 -989.049,E2 -989.049} C_VEL
LIN {X 0,Y 594.637,Z 342.188,A -85,B 0,C 180,E1 -989.345,E2 -989.345} C_VEL
LIN {X 0,Y 594.572,Z 355.258,A -85,B 0,C 180,E1 -989.79,E2 -989.79} C_VEL
LIN {X 0,Y 594.515,Z 367.096,A -85,B 0,C 180,E1 -990.34,E2 -990.34} C_VEL
LIN {X 0,Y 594.412,Z 378.437,A -85,B 0,C 180,E1 -991.017,E2 -991.017} C_VEL
LIN {X 0,Y 594.428,Z 388.656,A -85,B 0,C 180,E1 -991.78,E2 -991.78} C_VEL
LIN {X 0,Y 594.347,Z 397.086,A -85,B 0,C 180,E1 -992.543,E2 -992.543} C_VEL
LIN {X 0,Y 594.326,Z 404.879,A -85,B 0,C 180,E1 -993.391,E2 -993.391} C_VEL
LIN {X 0,Y 594.296,Z 412.523,A -85,B 0,C 180,E1 -994.409,E2 -994.409} C_VEL
LIN {X 0,Y 594.288,Z 418.685,A -85,B 0,C 180,E1 -995.429,E2 -995.429} C_VEL
LIN {X 0,Y 594.273,Z 424.148,A -85,B 0,C 180,E1 -996.583,E2 -996.583} C_VEL
LIN {X 0,Y 594.256,Z 427.398,A -85,B 0,C 180,E1 -997.475,E2 -997.475} C_VEL
LIN {X 0,Y 594.23,Z 429.359,A -85,B 0,C 180,E1 -998.16,E2 -998.16} C_VEL
LIN {X 0,Y 594.228,Z 430.905,A -85,B 0,C 180,E1 -998.845,E2 -998.845} C_VEL
LIN {X 0,Y 594.256,Z 432.001,A -85,B 0,C 180,E1 -999.531,E2 -999.531} C_VEL
LIN {X 0,Y 594.241,Z 432.975,A -85,B 0,C 180,E1 -1000.908,E2 -1000.908} C_VEL
LIN {X 0,Y 594.234,Z 432.867,A -85,B 0,C 180,E1 -1001.599,E2 -1001.599} C_VEL
LIN {X 0,Y 594.24,Z 432.31,A -85,B 0,C 180,E1 -1002.291,E2 -1002.291} C_VEL
LIN {X 0,Y 594.245,Z 431.352,A -85,B 0,C 180,E1 -1002.986,E2 -1002.986} C_VEL
LIN {X 0,Y 594.263,Z 428.853,A -85,B 0,C 180,E1 -1004.124,E2 -1004.124} C_VEL
LIN {X 0,Y 594.257,Z 425.798,A -85,B 0,C 180,E1 -1005.081,E2 -1005.081} C_VEL
LIN {X 0,Y 594.275,Z 421.356,A -85,B 0,C 180,E1 -1006.136,E2 -1006.136} C_VEL
LIN {X 0,Y 594.327,Z 415.627,A -85,B 0,C 180,E1 -1007.195,E2 -1007.195} C_VEL
LIN {X 0,Y 594.338,Z 408.376,A -85,B 0,C 180,E1 -1008.261,E2 -1008.261} C_VEL
LIN {X 0,Y 594.363,Z 399.163,A -85,B 0,C 180,E1 -1009.334,E2 -1009.334} C_VEL
LIN {X 0,Y 594.419,Z 389.619,A -85,B 0,C 180,E1 -1010.232,E2 -1010.232} C_VEL
LIN {X 0,Y 594.446,Z 379.398,A -85,B 0,C 180,E1 -1011.007,E2 -1011.007} C_VEL
LIN {X 0,Y 594.498,Z 368.392,A -85,B 0,C 180,E1 -1011.68,E2 -1011.68} C_VEL
LIN {X 0,Y 594.57,Z 357.076,A -85,B 0,C 180,E1 -1012.224,E2 -1012.224} C_VEL
LIN {X 0,Y 594.553,Z 344.413,A -85,B 0,C 180,E1 -1012.683,E2 -1012.683} C_VEL
LIN {X 0,Y 594.611,Z 331.321,A -85,B 0,C 180,E1 -1013.002,E2 -1013.002} C_VEL
LIN {X 0,Y 594.633,Z 311.192,A -85,B 0,C 180,E1 -1013.277,E2 -1013.277} C_VEL
LIN {X 0,Y 594.642,Z 224.459,A -85,B 0,C 180,E1 -1014.329,E2 -1014.329} C_VEL
LIN {X 0,Y 594.363,Z 222.555,A -85,B 0,C 180,E1 -1014.376,E2 -1014.376} C_VEL
LIN {X 0,Y 594.413,Z 207.463,A -85,B 0,C 180,E1 -1017.076,E2 -1017.076} C_VEL
LIN {X 0,Y 594.402,Z 195.441,A -85,B 0,C 180,E1 -1019.287,E2 -1019.287} C_VEL
LIN {X 0,Y 594.367,Z 195.448,A -85,B 0,C 180,E1 -1022.145,E2 -1022.145} C_VEL
LIN {X 0,Y 594.384,Z 195.447,A -85,B 0,C 180,E1 -1024.577,E2 -1024.577} C_VEL
LIN {X 0,Y 594.375,Z 195.442,A -85,B 0,C 180,E1 -1027.085,E2 -1027.085} C_VEL
LIN {X 0,Y 594.368,Z 195.445,A -85,B 0,C 180,E1 -1029.773,E2 -1029.773} C_VEL
LIN {X 0,Y 594.36,Z 195.451,A -85,B 0,C 180,E1 -1032.373,E2 -1032.373} C_VEL
LIN {X 0,Y 594.346,Z 195.445,A -85,B 0,C 180,E1 -1035.189,E2 -1035.189} C_VEL
LIN {X 0,Y 594.373,Z 195.445,A -85,B 0,C 180,E1 -1037.625,E2 -1037.625} C_VEL
LIN {X 0,Y 594.378,Z 195.447,A -85,B 0,C 180,E1 -1040.319,E2 -1040.319} C_VEL
LIN {X 0,Y 594.364,Z 195.442,A -85,B 0,C 180,E1 -1042.911,E2 -1042.911} C_VEL
LIN {X 0,Y 594.369,Z 195.451,A -85,B 0,C 180,E1 -1045.857,E2 -1045.857} C_VEL
LIN {X 0,Y 594.366,Z 195.443,A -85,B 0,C 180,E1 -1048.649,E2 -1048.649} C_VEL
LIN {X 0,Y 594.369,Z 195.442,A -85,B 0,C 180,E1 -1051.037,E2 -1051.037} C_VEL
LIN {X 0,Y 594.36,Z 195.45,A -85,B 0,C 180,E1 -1053.974,E2 -1053.974} C_VEL
LIN {X 0,Y 594.369,Z 195.443,A -85,B 0,C 180,E1 -1056.295,E2 -1056.295} C_VEL
LIN {X 0,Y 594.394,Z 195.442,A -85,B 0,C 180,E1 -1059.224,E2 -1059.224} C_VEL
LIN {X 0,Y 594.351,Z 195.447,A -85,B 0,C 180,E1 -1062.095,E2 -1062.095} C_VEL
LIN {X 0,Y 594.342,Z 195.446,A -85,B 0,C 180,E1 -1064.218,E2 -1064.218} C_VEL
LIN {X 0,Y 594.347,Z 195.445,A -85,B 0,C 180,E1 -1066.32,E2 -1066.32} C_VEL
LIN {X 0,Y 594.364,Z 195.447,A -85,B 0,C 180,E1 -1069.094,E2 -1069.094} C_VEL
LIN {X 0,Y 594.38,Z 195.444,A -85,B 0,C 180,E1 -1071.843,E2 -1071.843} C_VEL
LIN {X 0,Y 594.329,Z 195.449,A -85,B 0,C 180,E1 -1073.891,E2 -1073.891} C_VEL
LIN {X 0,Y 594.316,Z 195.45,A -85,B 0,C 180,E1 -1075.931,E2 -1075.931} C_VEL
LIN {X 0,Y 594.346,Z 195.445,A -85,B 0,C 180,E1 -1077.967,E2 -1077.967} C_VEL
LIN {X 0,Y 594.36,Z 195.443,A -85,B 0,C 180,E1 -1080,E2 -1080} C_VEL
LIN {X 0,Y 594.377,Z 195.444,A -85,B 0,C 180,E1 -1082.711,E2 -1082.711} C_VEL
LIN {X 0,Y 594.365,Z 195.447,A -85,B 0,C 180,E1 -1085.428,E2 -1085.428} C_VEL
LIN {X 0,Y 594.36,Z 195.446,A -85,B 0,C 180,E1 -1087.474,E2 -1087.474} C_VEL
LIN {X 0,Y 594.348,Z 195.445,A -85,B 0,C 180,E1 -1090.217,E2 -1090.217} C_VEL
LIN {X 0,Y 594.345,Z 195.446,A -85,B 0,C 180,E1 -1092.289,E2 -1092.289} C_VEL
LIN {X 0,Y 594.334,Z 195.453,A -85,B 0,C 180,E1 -1095.079,E2 -1095.079} C_VEL
LIN {X 0,Y 594.348,Z 195.449,A -85,B 0,C 180,E1 -1097.195,E2 -1097.195} C_VEL
LIN {X 0,Y 594.332,Z 195.447,A -85,B 0,C 180,E1 -1100.055,E2 -1100.055} C_VEL
LIN {X 0,Y 594.326,Z 195.453,A -85,B 0,C 180,E1 -1102.969,E2 -1102.969} C_VEL
LIN {X 0,Y 594.321,Z 195.45,A -85,B 0,C 180,E1 -1105.196,E2 -1105.196} C_VEL
LIN {X 0,Y 594.312,Z 195.449,A -85,B 0,C 180,E1 -1107.521,E2 -1107.521} C_VEL
LIN {X 0,Y 594.329,Z 195.447,A -85,B 0,C 180,E1 -1109.779,E2 -1109.779} C_VEL
LIN {X 0,Y 594.346,Z 195.449,A -85,B 0,C 180,E1 -1112.149,E2 -1112.149} C_VEL
LIN {X 0,Y 594.35,Z 195.453,A -85,B 0,C 180,E1 -1114.582,E2 -1114.582} C_VEL
LIN {X 0,Y 594.36,Z 195.443,A -85,B 0,C 180,E1 -1117.61,E2 -1117.61} C_VEL
LIN {X 0,Y 594.361,Z 195.45,A -85,B 0,C 180,E1 -1120.568,E2 -1120.568} C_VEL
LIN {X 0,Y 594.338,Z 195.446,A -85,B 0,C 180,E1 -1123.302,E2 -1123.302} C_VEL
LIN {X 0,Y 594.343,Z 195.454,A -85,B 0,C 180,E1 -1126.163,E2 -1126.163} C_VEL
LIN {X 0,Y 594.351,Z 195.444,A -85,B 0,C 180,E1 -1129.181,E2 -1129.181} C_VEL
LIN {X 0,Y 594.367,Z 195.452,A -85,B 0,C 180,E1 -1132.061,E2 -1132.061} C_VEL
LIN {X 0,Y 594.341,Z 195.447,A -85,B 0,C 180,E1 -1134.678,E2 -1134.678} C_VEL
LIN {X 0,Y 594.366,Z 195.442,A -85,B 0,C 180,E1 -1137.091,E2 -1137.091} C_VEL
LIN {X 0,Y 594.379,Z 195.447,A -85,B 0,C 180,E1 -1139.673,E2 -1139.673} C_VEL
LIN {X 0,Y 594.371,Z 195.443,A -85,B 0,C 180,E1 -1142.54,E2 -1142.54} C_VEL
LIN {X 0,Y 594.397,Z 195.446,A -85,B 0,C 180,E1 -1145.565,E2 -1145.565} C_VEL
LIN {X 0,Y 594.361,Z 195.489,A -85,B 0,C 180,E1 -1146.573,E2 -1146.573} C_VEL
LIN {X 0,Y 594.786,Z 199.667,A -85,B 0,C 180,E1 -1147.169,E2 -1147.169} C_VEL
LIN {X 0,Y 594.669,Z 220.085,A -85,B 0,C 180,E1 -1149.957,E2 -1149.957} C_VEL
LIN {X 0,Y 594.564,Z 240.027,A -85,B 0,C 180,E1 -1152.635,E2 -1152.635} C_VEL
LIN {X 0,Y 594.472,Z 261.299,A -85,B 0,C 180,E1 -1155.45,E2 -1155.45} C_VEL
LIN {X 0,Y 594.434,Z 270.439,A -85,B 0,C 180,E1 -1156.649,E2 -1156.649} C_VEL
LIN {X 0,Y 594.732,Z 276.509,A -85,B 0,C 180,E1 -1156.743,E2 -1156.743} C_VEL
LIN {X 0,Y 594.657,Z 378.941,A -85,B 0,C 180,E1 -1157.999,E2 -1157.999} C_VEL
LIN {X 0,Y 594.631,Z 392.213,A -85,B 0,C 180,E1 -1158.301,E2 -1158.301} C_VEL
LIN {X 0,Y 594.597,Z 404.43,A -85,B 0,C 180,E1 -1158.713,E2 -1158.713} C_VEL
LIN {X 0,Y 594.528,Z 416.627,A -85,B 0,C 180,E1 -1159.27,E2 -1159.27} C_VEL
LIN {X 0,Y 594.48,Z 428.196,A -85,B 0,C 180,E1 -1159.957,E2 -1159.957} C_VEL
LIN {X 0,Y 594.414,Z 438.592,A -85,B 0,C 180,E1 -1160.729,E2 -1160.729} C_VEL
LIN {X 0,Y 594.383,Z 447.107,A -85,B 0,C 180,E1 -1161.5,E2 -1161.5} C_VEL
LIN {X 0,Y 594.347,Z 454.956,A -85,B 0,C 180,E1 -1162.355,E2 -1162.355} C_VEL
LIN {X 0,Y 594.283,Z 462.811,A -85,B 0,C 180,E1 -1163.408,E2 -1163.408} C_VEL
LIN {X 0,Y 594.289,Z 469.676,A -85,B 0,C 180,E1 -1164.571,E2 -1164.571} C_VEL
LIN {X 0,Y 594.27,Z 474.368,A -85,B 0,C 180,E1 -1165.59,E2 -1165.59} C_VEL
LIN {X 0,Y 594.267,Z 477.953,A -85,B 0,C 180,E1 -1166.609,E2 -1166.609} C_VEL
LIN {X 0,Y 594.226,Z 479.806,A -85,B 0,C 180,E1 -1167.287,E2 -1167.287} C_VEL
LIN {X 0,Y 594.242,Z 481.199,A -85,B 0,C 180,E1 -1167.966,E2 -1167.966} C_VEL
LIN {X 0,Y 594.239,Z 482.783,A -85,B 0,C 180,E1 -1169.321,E2 -1169.321} C_VEL
LIN {X 0,Y 594.236,Z 483,A -85,B 0,C 180,E1 -1169.999,E2 -1169.999} C_VEL
LIN {X 0,Y 594.247,Z 482.187,A -85,B 0,C 180,E1 -1171.354,E2 -1171.354} C_VEL
LIN {X 0,Y 594.242,Z 481.204,A -85,B 0,C 180,E1 -1172.032,E2 -1172.032} C_VEL
LIN {X 0,Y 594.225,Z 479.813,A -85,B 0,C 180,E1 -1172.71,E2 -1172.71} C_VEL
LIN {X 0,Y 594.289,Z 476.901,A -85,B 0,C 180,E1 -1173.728,E2 -1173.728} C_VEL
LIN {X 0,Y 594.241,Z 472.957,A -85,B 0,C 180,E1 -1174.747,E2 -1174.747} C_VEL
LIN {X 0,Y 594.304,Z 466.889,A -85,B 0,C 180,E1 -1175.937,E2 -1175.937} C_VEL
LIN {X 0,Y 594.31,Z 460.251,A -85,B 0,C 180,E1 -1176.96,E2 -1176.96} C_VEL
LIN {X 0,Y 594.358,Z 452.008,A -85,B 0,C 180,E1 -1177.984,E2 -1177.984} C_VEL
LIN {X 0,Y 594.381,Z 443.561,A -85,B 0,C 180,E1 -1178.84,E2 -1178.84} C_VEL
LIN {X 0,Y 594.433,Z 433.125,A -85,B 0,C 180,E1 -1179.697,E2 -1179.697} C_VEL
LIN {X 0,Y 594.485,Z 422.797,A -85,B 0,C 180,E1 -1180.384,E2 -1180.384} C_VEL
LIN {X 0,Y 594.558,Z 411.724,A -85,B 0,C 180,E1 -1180.973,E2 -1180.973} C_VEL
LIN {X 0,Y 594.573,Z 399.77,A -85,B 0,C 180,E1 -1181.462,E2 -1181.462} C_VEL
LIN {X 0,Y 594.635,Z 386.455,A -85,B 0,C 180,E1 -1181.848,E2 -1181.848} C_VEL
LIN {X 0,Y 594.692,Z 373.268,A -85,B 0,C 180,E1 -1182.085,E2 -1182.085} C_VEL
LIN {X 0,Y 594.626,Z 272.029,A -85,B 0,C 180,E1 -1183.314,E2 -1183.314} C_VEL
LIN {X 0,Y 594.433,Z 270.459,A -85,B 0,C 180,E1 -1183.349,E2 -1183.349} C_VEL
LIN {X 0,Y 594.537,Z 248.024,A -85,B 0,C 180,E1 -1186.302,E2 -1186.302} C_VEL
LIN {X 0,Y 594.618,Z 227.112,A -85,B 0,C 180,E1 -1189.095,E2 -1189.095} C_VEL
LIN {X 0,Y 594.759,Z 206.81,A -85,B 0,C 180,E1 -1191.849,E2 -1191.849} C_VEL
LIN {X 0,Y 594.738,Z 197.504,A -85,B 0,C 180,E1 -1193.132,E2 -1193.132} C_VEL
LIN {X 0,Y 594.364,Z 195.448,A -85,B 0,C 180,E1 -1193.47,E2 -1193.47} C_VEL
LIN {X 0,Y 594.384,Z 195.449,A -85,B 0,C 180,E1 -1196.022,E2 -1196.022} C_VEL
LIN {X 0,Y 594.36,Z 195.443,A -85,B 0,C 180,E1 -1198.995,E2 -1198.995} C_VEL
LIN {X 0,Y 594.36,Z 195.446,A -85,B 0,C 180,E1 -1201.64,E2 -1201.64} C_VEL
LIN {X 0,Y 594.367,Z 195.444,A -85,B 0,C 180,E1 -1204.575,E2 -1204.575} C_VEL
LIN {X 0,Y 594.358,Z 195.443,A -85,B 0,C 180,E1 -1207.083,E2 -1207.083} C_VEL
LIN {X 0,Y 594.354,Z 195.452,A -85,B 0,C 180,E1 -1209.771,E2 -1209.771} C_VEL
LIN {X 0,Y 594.338,Z 195.448,A -85,B 0,C 180,E1 -1212.371,E2 -1212.371} C_VEL
LIN {X 0,Y 594.327,Z 195.448,A -85,B 0,C 180,E1 -1215.187,E2 -1215.187} C_VEL
LIN {X 0,Y 594.365,Z 195.45,A -85,B 0,C 180,E1 -1217.624,E2 -1217.624} C_VEL
LIN {X 0,Y 594.363,Z 195.444,A -85,B 0,C 180,E1 -1220.318,E2 -1220.318} C_VEL
LIN {X 0,Y 594.346,Z 195.445,A -85,B 0,C 180,E1 -1222.91,E2 -1222.91} C_VEL
LIN {X 0,Y 594.349,Z 195.451,A -85,B 0,C 180,E1 -1225.856,E2 -1225.856} C_VEL
LIN {X 0,Y 594.351,Z 195.445,A -85,B 0,C 180,E1 -1228.35,E2 -1228.35} C_VEL
LIN {X 0,Y 594.376,Z 195.443,A -85,B 0,C 180,E1 -1231.031,E2 -1231.031} C_VEL
LIN {X 0,Y 594.342,Z 195.448,A -85,B 0,C 180,E1 -1233.972,E2 -1233.972} C_VEL
LIN {X 0,Y 594.365,Z 195.446,A -85,B 0,C 180,E1 -1237.033,E2 -1237.033} C_VEL
LIN {X 0,Y 594.338,Z 195.448,A -85,B 0,C 180,E1 -1239.945,E2 -1239.945} C_VEL
LIN {X 0,Y 594.334,Z 195.447,A -85,B 0,C 180,E1 -1242.094,E2 -1242.094} C_VEL
LIN {X 0,Y 594.325,Z 195.447,A -85,B 0,C 180,E1 -1244.218,E2 -1244.218} C_VEL
LIN {X 0,Y 594.353,Z 195.45,A -85,B 0,C 180,E1 -1247.017,E2 -1247.017} C_VEL
LIN {X 0,Y 594.374,Z 195.449,A -85,B 0,C 180,E1 -1249.095,E2 -1249.095} C_VEL
LIN {X 0,Y 594.359,Z 195.444,A -85,B 0,C 180,E1 -1251.843,E2 -1251.843} C_VEL
LIN {X 0,Y 594.311,Z 195.45,A -85,B 0,C 180,E1 -1253.891,E2 -1253.891} C_VEL
LIN {X 0,Y 594.341,Z 195.448,A -85,B 0,C 180,E1 -1256.611,E2 -1256.611} C_VEL
LIN {X 0,Y 594.383,Z 195.446,A -85,B 0,C 180,E1 -1259.323,E2 -1259.323} C_VEL
LIN {X 0,Y 594.326,Z 195.447,A -85,B 0,C 180,E1 -1262.033,E2 -1262.033} C_VEL
LIN {X 0,Y 594.351,Z 195.451,A -85,B 0,C 180,E1 -1264.748,E2 -1264.748} C_VEL
LIN {X 0,Y 594.359,Z 195.445,A -85,B 0,C 180,E1 -1267.474,E2 -1267.474} C_VEL
LIN {X 0,Y 594.339,Z 195.447,A -85,B 0,C 180,E1 -1270.217,E2 -1270.217} C_VEL
LIN {X 0,Y 594.336,Z 195.448,A -85,B 0,C 180,E1 -1272.404,E2 -1272.404} C_VEL
LIN {X 0,Y 594.328,Z 195.452,A -85,B 0,C 180,E1 -1275.079,E2 -1275.079} C_VEL
LIN {X 0,Y 594.314,Z 195.451,A -85,B 0,C 180,E1 -1275.358,E2 -1275.358} C_VEL
LIN {X 0,Y 593.642,Z 195.534,A -85,B 0,C 180,E1 -1275.924,E2 -1275.924} C_VEL
LIN {X 0,Y 590.784,Z 195.897,A -85,B 0,C 180,E1 -1276.842,E2 -1276.842} C_VEL
LIN {X 0,Y 588.379,Z 196.193,A -85,B 0,C 180,E1 -1277.581,E2 -1277.581} C_VEL
LIN {X 0,Y 587.359,Z 196.317,A -85,B 0,C 180,E1 -1278.151,E2 -1278.151} C_VEL
LIN {X 0,Y 587.282,Z 196.327,A -85,B 0,C 180,E1 -1278.344,E2 -1278.344} C_VEL
LIN {X 0,Y 587.303,Z 196.326,A -85,B 0,C 180,E1 -1281.048,E2 -1281.048} C_VEL
LIN {X 0,Y 587.313,Z 196.322,A -85,B 0,C 180,E1 -1283.259,E2 -1283.259} C_VEL
LIN {X 0,Y 587.31,Z 196.326,A -85,B 0,C 180,E1 -1286.28,E2 -1286.28} C_VEL
LIN {X 0,Y 587.328,Z 196.321,A -85,B 0,C 180,E1 -1289.142,E2 -1289.142} C_VEL
LIN {X 0,Y 587.315,Z 196.322,A -85,B 0,C 180,E1 -1291.842,E2 -1291.842} C_VEL
LIN {X 0,Y 587.317,Z 196.329,A -85,B 0,C 180,E1 -1294.354,E2 -1294.354} C_VEL
LIN {X 0,Y 587.31,Z 196.326,A -85,B 0,C 180,E1 -1296.75,E2 -1296.75} C_VEL
LIN {X 0,Y 587.294,Z 196.323,A -85,B 0,C 180,E1 -1299.364,E2 -1299.364} C_VEL
LIN {X 0,Y 587.329,Z 196.326,A -85,B 0,C 180,E1 -1302.115,E2 -1302.115} C_VEL
LIN {X 0,Y 587.28,Z 196.325,A -85,B 0,C 180,E1 -1305.093,E2 -1305.093} C_VEL
LIN {X 0,Y 587.322,Z 196.325,A -85,B 0,C 180,E1 -1307.932,E2 -1307.932} C_VEL
LIN {X 0,Y 587.3,Z 196.323,A -85,B 0,C 180,E1 -1311.063,E2 -1311.063} C_VEL
LIN {X 0,Y 587.327,Z 196.319,A -85,B 0,C 180,E1 -1313.296,E2 -1313.296} C_VEL
LIN {X 0,Y 587.339,Z 196.323,A -85,B 0,C 180,E1 -1315.784,E2 -1315.784} C_VEL
LIN {X 0,Y 587.32,Z 196.327,A -85,B 0,C 180,E1 -1318.235,E2 -1318.235} C_VEL
LIN {X 0,Y 587.33,Z 196.319,A -85,B 0,C 180,E1 -1320.871,E2 -1320.871} C_VEL
LIN {X 0,Y 587.348,Z 196.325,A -85,B 0,C 180,E1 -1323.822,E2 -1323.822} C_VEL
LIN {X 0,Y 587.322,Z 196.328,A -85,B 0,C 180,E1 -1325.997,E2 -1325.997} C_VEL
LIN {X 0,Y 587.307,Z 196.326,A -85,B 0,C 180,E1 -1328.229,E2 -1328.229} C_VEL
LIN {X 0,Y 587.328,Z 196.32,A -85,B 0,C 180,E1 -1331.154,E2 -1331.154} C_VEL
LIN {X 0,Y 587.304,Z 196.327,A -85,B 0,C 180,E1 -1334.027,E2 -1334.027} C_VEL
LIN {X 0,Y 587.35,Z 196.319,A -85,B 0,C 180,E1 -1336.157,E2 -1336.157} C_VEL
LIN {X 0,Y 587.337,Z 196.319,A -85,B 0,C 180,E1 -1338.965,E2 -1338.965} C_VEL
LIN {X 0,Y 587.362,Z 196.324,A -85,B 0,C 180,E1 -1341.747,E2 -1341.747} C_VEL
LIN {X 0,Y 587.319,Z 196.396,A -85,B 0,C 180,E1 -1342.784,E2 -1342.784} C_VEL
LIN {X 0,Y 587.418,Z 205.777,A -85,B 0,C 180,E1 -1344.509,E2 -1344.509} C_VEL
LIN {X 0,Y 587.366,Z 221.878,A -85,B 0,C 180,E1 -1347.43,E2 -1347.43} C_VEL
LIN {X 0,Y 587.357,Z 222.593,A -85,B 0,C 180,E1 -1347.558,E2 -1347.558} C_VEL
LIN {X 0,Y 587.849,Z 227.86,A -85,B 0,C 180,E1 -1347.646,E2 -1347.646} C_VEL
LIN {X 0,Y 587.693,Z 329.464,A -85,B 0,C 180,E1 -1348.909,E2 -1348.909} C_VEL
LIN {X 0,Y 587.677,Z 343.081,A -85,B 0,C 180,E1 -1349.23,E2 -1349.23} C_VEL
LIN {X 0,Y 587.603,Z 355.369,A -85,B 0,C 180,E1 -1349.659,E2 -1349.659} C_VEL
LIN {X 0,Y 587.531,Z 366.393,A -85,B 0,C 180,E1 -1350.173,E2 -1350.173} C_VEL
LIN {X 0,Y 587.389,Z 377.878,A -85,B 0,C 180,E1 -1350.858,E2 -1350.858} C_VEL
LIN {X 0,Y 587.391,Z 388.193,A -85,B 0,C 180,E1 -1351.629,E2 -1351.629} C_VEL
LIN {X 0,Y 587.301,Z 396.695,A -85,B 0,C 180,E1 -1352.401,E2 -1352.401} C_VEL
LIN {X 0,Y 587.271,Z 404.551,A -85,B 0,C 180,E1 -1353.26,E2 -1353.26} C_VEL
LIN {X 0,Y 587.231,Z 412.274,A -85,B 0,C 180,E1 -1354.291,E2 -1354.291} C_VEL
LIN {X 0,Y 587.21,Z 419.388,A -85,B 0,C 180,E1 -1355.495,E2 -1355.495} C_VEL
LIN {X 0,Y 587.197,Z 424.363,A -85,B 0,C 180,E1 -1356.581,E2 -1356.581} C_VEL
LIN {X 0,Y 587.152,Z 427.812,A -85,B 0,C 180,E1 -1357.566,E2 -1357.566} C_VEL
LIN {X 0,Y 587.14,Z 429.705,A -85,B 0,C 180,E1 -1358.259,E2 -1358.259} C_VEL
LIN {X 0,Y 587.128,Z 431.144,A -85,B 0,C 180,E1 -1358.953,E2 -1358.953} C_VEL
LIN {X 0,Y 587.151,Z 432.156,A -85,B 0,C 180,E1 -1359.647,E2 -1359.647} C_VEL
LIN {X 0,Y 587.168,Z 433,A -85,B 0,C 180,E1 -1361.041,E2 -1361.041} C_VEL
LIN {X 0,Y 587.155,Z 432.778,A -85,B 0,C 180,E1 -1361.741,E2 -1361.741} C_VEL
LIN {X 0,Y 587.161,Z 432.156,A -85,B 0,C 180,E1 -1362.442,E2 -1362.442} C_VEL
LIN {X 0,Y 587.146,Z 431.13,A -85,B 0,C 180,E1 -1363.146,E2 -1363.146} C_VEL
LIN {X 0,Y 587.161,Z 428.803,A -85,B 0,C 180,E1 -1364.18,E2 -1364.18} C_VEL
LIN {X 0,Y 587.173,Z 425.303,A -85,B 0,C 180,E1 -1365.267,E2 -1365.267} C_VEL
LIN {X 0,Y 587.175,Z 420.706,A -85,B 0,C 180,E1 -1366.336,E2 -1366.336} C_VEL
LIN {X 0,Y 587.245,Z 414.799,A -85,B 0,C 180,E1 -1367.409,E2 -1367.409} C_VEL
LIN {X 0,Y 587.247,Z 407.275,A -85,B 0,C 180,E1 -1368.49,E2 -1368.49} C_VEL
LIN {X 0,Y 587.362,Z 397.844,A -85,B 0,C 180,E1 -1369.574,E2 -1369.574} C_VEL
LIN {X 0,Y 587.38,Z 387.895,A -85,B 0,C 180,E1 -1370.485,E2 -1370.485} C_VEL
LIN {X 0,Y 587.438,Z 377.261,A -85,B 0,C 180,E1 -1371.273,E2 -1371.273} C_VEL
LIN {X 0,Y 587.517,Z 365.761,A -85,B 0,C 180,E1 -1371.95,E2 -1371.95} C_VEL
LIN {X 0,Y 587.589,Z 353.545,A -85,B 0,C 180,E1 -1372.503,E2 -1372.503} C_VEL
LIN {X 0,Y 587.65,Z 341.023,A -85,B 0,C 180,E1 -1372.919,E2 -1372.919} C_VEL
LIN {X 0,Y 587.675,Z 328.384,A -85,B 0,C 180,E1 -1373.201,E2 -1373.201} C_VEL
LIN {X 0,Y 587.782,Z 225.399,A -85,B 0,C 180,E1 -1374.476,E2 -1374.476} C_VEL
LIN {X 0,Y 587.302,Z 222.592,A -85,B 0,C 180,E1 -1374.533,E2 -1374.533} C_VEL
LIN {X 0,Y 587.384,Z 206.925,A -85,B 0,C 180,E1 -1377.372,E2 -1377.372} C_VEL
LIN {X 0,Y 587.374,Z 196.317,A -85,B 0,C 180,E1 -1379.339,E2 -1379.339} C_VEL
LIN {X 0,Y 587.343,Z 196.32,A -85,B 0,C 180,E1 -1381.835,E2 -1381.835} C_VEL
LIN {X 0,Y 587.347,Z 196.327,A -85,B 0,C 180,E1 -1384.347,E2 -1384.347} C_VEL
LIN {X 0,Y 587.343,Z 196.322,A -85,B 0,C 180,E1 -1386.745,E2 -1386.745} C_VEL
LIN {X 0,Y 587.336,Z 196.319,A -85,B 0,C 180,E1 -1389.357,E2 -1389.357} C_VEL
LIN {X 0,Y 587.321,Z 196.329,A -85,B 0,C 180,E1 -1392.106,E2 -1392.106} C_VEL
LIN {X 0,Y 587.299,Z 196.324,A -85,B 0,C 180,E1 -1394.909,E2 -1394.909} C_VEL
LIN {X 0,Y 587.334,Z 196.326,A -85,B 0,C 180,E1 -1397.925,E2 -1397.925} C_VEL
LIN {X 0,Y 587.316,Z 196.321,A -85,B 0,C 180,E1 -1401.056,E2 -1401.056} C_VEL
LIN {X 0,Y 587.332,Z 196.319,A -85,B 0,C 180,E1 -1403.289,E2 -1403.289} C_VEL
LIN {X 0,Y 587.35,Z 196.324,A -85,B 0,C 180,E1 -1405.779,E2 -1405.779} C_VEL
LIN {X 0,Y 587.333,Z 196.323,A -85,B 0,C 180,E1 -1408.23,E2 -1408.23} C_VEL
LIN {X 0,Y 587.332,Z 196.319,A -85,B 0,C 180,E1 -1410.862,E2 -1410.862} C_VEL
LIN {X 0,Y 587.331,Z 196.328,A -85,B 0,C 180,E1 -1413.816,E2 -1413.816} C_VEL
LIN {X 0,Y 587.338,Z 196.317,A -85,B 0,C 180,E1 -1416.742,E2 -1416.742} C_VEL
LIN {X 0,Y 587.314,Z 196.33,A -85,B 0,C 180,E1 -1419.694,E2 -1419.694} C_VEL
LIN {X 0,Y 587.305,Z 196.328,A -85,B 0,C 180,E1 -1421.873,E2 -1421.873} C_VEL
LIN {X 0,Y 587.306,Z 196.324,A -85,B 0,C 180,E1 -1424.024,E2 -1424.024} C_VEL
LIN {X 0,Y 587.33,Z 196.32,A -85,B 0,C 180,E1 -1426.153,E2 -1426.153} C_VEL
LIN {X 0,Y 587.324,Z 196.322,A -85,B 0,C 180,E1 -1428.962,E2 -1428.962} C_VEL
LIN {X 0,Y 587.336,Z 196.322,A -85,B 0,C 180,E1 -1431.744,E2 -1431.744} C_VEL
LIN {X 0,Y 587.289,Z 196.326,A -85,B 0,C 180,E1 -1433.817,E2 -1433.817} C_VEL
LIN {X 0,Y 587.273,Z 196.328,A -85,B 0,C 180,E1 -1435.882,E2 -1435.882} C_VEL
LIN {X 0,Y 587.318,Z 196.32,A -85,B 0,C 180,E1 -1437.943,E2 -1437.943} C_VEL
LIN {X 0,Y 587.33,Z 196.319,A -85,B 0,C 180,E1 -1440,E2 -1440} C_VEL
LIN {X 0,Y 587.342,Z 196.321,A -85,B 0,C 180,E1 -1442.743,E2 -1442.743} C_VEL
LIN {X 0,Y 587.327,Z 196.323,A -85,B 0,C 180,E1 -1445.493,E2 -1445.493} C_VEL
LIN {X 0,Y 587.29,Z 196.324,A -85,B 0,C 180,E1 -1448.256,E2 -1448.256} C_VEL
LIN {X 0,Y 587.373,Z 196.32,A -85,B 0,C 180,E1 -1451.167,E2 -1451.167} C_VEL
LIN {X 0,Y 587.298,Z 196.327,A -85,B 0,C 180,E1 -1454.554,E2 -1454.554} C_VEL
LIN {X 0,Y 587.306,Z 196.323,A -85,B 0,C 180,E1 -1457.407,E2 -1457.407} C_VEL
LIN {X 0,Y 587.272,Z 196.327,A -85,B 0,C 180,E1 -1459.578,E2 -1459.578} C_VEL
LIN {X 0,Y 587.279,Z 196.325,A -85,B 0,C 180,E1 -1461.776,E2 -1461.776} C_VEL
LIN {X 0,Y 587.31,Z 196.33,A -85,B 0,C 180,E1 -1464.76,E2 -1464.76} C_VEL
LIN {X 0,Y 587.271,Z 196.326,A -85,B 0,C 180,E1 -1467.686,E2 -1467.686} C_VEL
LIN {X 0,Y 587.286,Z 196.328,A -85,B 0,C 180,E1 -1470.173,E2 -1470.173} C_VEL
LIN {X 0,Y 587.314,Z 196.33,A -85,B 0,C 180,E1 -1472.581,E2 -1472.581} C_VEL
LIN {X 0,Y 587.296,Z 196.325,A -85,B 0,C 180,E1 -1475.058,E2 -1475.058} C_VEL
LIN {X 0,Y 587.312,Z 196.322,A -85,B 0,C 180,E1 -1477.84,E2 -1477.84} C_VEL
LIN {X 0,Y 587.295,Z 196.331,A -85,B 0,C 180,E1 -1480.256,E2 -1480.256} C_VEL
LIN {X 0,Y 587.303,Z 196.323,A -85,B 0,C 180,E1 -1483.008,E2 -1483.008} C_VEL
LIN {X 0,Y 587.295,Z 196.33,A -85,B 0,C 180,E1 -1486.05,E2 -1486.05} C_VEL
LIN {X 0,Y 587.317,Z 196.321,A -85,B 0,C 180,E1 -1488.927,E2 -1488.927} C_VEL
LIN {X 0,Y 587.305,Z 196.324,A -85,B 0,C 180,E1 -1491.522,E2 -1491.522} C_VEL
LIN {X 0,Y 587.293,Z 196.333,A -85,B 0,C 180,E1 -1494.103,E2 -1494.103} C_VEL
LIN {X 0,Y 587.329,Z 196.319,A -85,B 0,C 180,E1 -1496.89,E2 -1496.89} C_VEL
LIN {X 0,Y 587.326,Z 196.328,A -85,B 0,C 180,E1 -1499.831,E2 -1499.831} C_VEL
LIN {X 0,Y 587.3,Z 196.327,A -85,B 0,C 180,E1 -1502.317,E2 -1502.317} C_VEL
LIN {X 0,Y 587.346,Z 196.32,A -85,B 0,C 180,E1 -1505.242,E2 -1505.242} C_VEL
LIN {X 0,Y 587.343,Z 196.385,A -85,B 0,C 180,E1 -1506.416,E2 -1506.416} C_VEL
LIN {X 0,Y 587.882,Z 200.503,A -85,B 0,C 180,E1 -1507.002,E2 -1507.002} C_VEL
LIN {X 0,Y 587.761,Z 220.085,A -85,B 0,C 180,E1 -1509.711,E2 -1509.711} C_VEL
LIN {X 0,Y 587.575,Z 241.356,A -85,B 0,C 180,E1 -1512.601,E2 -1512.601} C_VEL
LIN {X 0,Y 587.475,Z 261.299,A -85,B 0,C 180,E1 -1515.273,E2 -1515.273} C_VEL
LIN {X 0,Y 587.402,Z 270.439,A -85,B 0,C 180,E1 -1516.486,E2 -1516.486} C_VEL
LIN {X 0,Y 587.84,Z 274.721,A -85,B 0,C 180,E1 -1516.562,E2 -1516.562} C_VEL
LIN {X 0,Y 587.72,Z 378.941,A -85,B 0,C 180,E1 -1517.855,E2 -1517.855} C_VEL
LIN {X 0,Y 587.681,Z 392.214,A -85,B 0,C 180,E1 -1518.16,E2 -1518.16} C_VEL
LIN {X 0,Y 587.629,Z 404.6,A -85,B 0,C 180,E1 -1518.584,E2 -1518.584} C_VEL
LIN {X 0,Y 587.53,Z 416.626,A -85,B 0,C 180,E1 -1519.14,E2 -1519.14} C_VEL
LIN {X 0,Y 587.468,Z 428.198,A -85,B 0,C 180,E1 -1519.836,E2 -1519.836} C_VEL
LIN {X 0,Y 587.394,Z 438.594,A -85,B 0,C 180,E1 -1520.617,E2 -1520.617} C_VEL
LIN {X 0,Y 587.322,Z 447.108,A -85,B 0,C 180,E1 -1521.397,E2 -1521.397} C_VEL
LIN {X 0,Y 587.274,Z 454.956,A -85,B 0,C 180,E1 -1522.262,E2 -1522.262} C_VEL
LIN {X 0,Y 587.231,Z 461.465,A -85,B 0,C 180,E1 -1523.126,E2 -1523.126} C_VEL
LIN {X 0,Y 587.236,Z 467.863,A -85,B 0,C 180,E1 -1524.161,E2 -1524.161} C_VEL
LIN {X 0,Y 587.147,Z 472.946,A -85,B 0,C 180,E1 -1525.193,E2 -1525.193} C_VEL
LIN {X 0,Y 587.213,Z 476.893,A -85,B 0,C 180,E1 -1526.225,E2 -1526.225} C_VEL
LIN {X 0,Y 587.132,Z 479.806,A -85,B 0,C 180,E1 -1527.255,E2 -1527.255} C_VEL
LIN {X 0,Y 587.141,Z 481.198,A -85,B 0,C 180,E1 -1527.941,E2 -1527.941} C_VEL
LIN {X 0,Y 587.14,Z 482.784,A -85,B 0,C 180,E1 -1529.313,E2 -1529.313} C_VEL
LIN {X 0,Y 587.137,Z 483,A -85,B 0,C 180,E1 -1529.999,E2 -1529.999} C_VEL
LIN {X 0,Y 587.147,Z 482.187,A -85,B 0,C 180,E1 -1531.37,E2 -1531.37} C_VEL
LIN {X 0,Y 587.141,Z 481.203,A -85,B 0,C 180,E1 -1532.056,E2 -1532.056} C_VEL
LIN {X 0,Y 587.132,Z 479.813,A -85,B 0,C 180,E1 -1532.743,E2 -1532.743} C_VEL
LIN {X 0,Y 587.213,Z 476.901,A -85,B 0,C 180,E1 -1533.773,E2 -1533.773} C_VEL
LIN {X 0,Y 587.147,Z 472.957,A -85,B 0,C 180,E1 -1534.805,E2 -1534.805} C_VEL
LIN {X 0,Y 587.236,Z 467.877,A -85,B 0,C 180,E1 -1535.837,E2 -1535.837} C_VEL
LIN {X 0,Y 587.23,Z 461.483,A -85,B 0,C 180,E1 -1536.872,E2 -1536.872} C_VEL
LIN {X 0,Y 587.286,Z 453.496,A -85,B 0,C 180,E1 -1537.908,E2 -1537.908} C_VEL
LIN {X 0,Y 587.335,Z 445.359,A -85,B 0,C 180,E1 -1538.773,E2 -1538.773} C_VEL
LIN {X 0,Y 587.391,Z 435.43,A -85,B 0,C 180,E1 -1539.641,E2 -1539.641} C_VEL
LIN {X 0,Y 587.481,Z 424.211,A -85,B 0,C 180,E1 -1540.422,E2 -1540.422} C_VEL
LIN {X 0,Y 587.58,Z 412.557,A -85,B 0,C 180,E1 -1541.064,E2 -1541.064} C_VEL
LIN {X 0,Y 587.609,Z 400.022,A -85,B 0,C 180,E1 -1541.592,E2 -1541.592} C_VEL
LIN {X 0,Y 587.688,Z 387.368,A -85,B 0,C 180,E1 -1541.968,E2 -1541.968} C_VEL
LIN {X 0,Y 587.75,Z 374.775,A -85,B 0,C 180,E1 -1542.208,E2 -1542.208} C_VEL
LIN {X 0,Y 587.719,Z 272.7,A -85,B 0,C 180,E1 -1543.465,E2 -1543.465} C_VEL
LIN {X 0,Y 587.4,Z 270.459,A -85,B 0,C 180,E1 -1543.511,E2 -1543.511} C_VEL
LIN {X 0,Y 587.556,Z 249.353,A -85,B 0,C 180,E1 -1546.322,E2 -1546.322} C_VEL
LIN {X 0,Y 587.672,Z 227.465,A -85,B 0,C 180,E1 -1549.281,E2 -1549.281} C_VEL
LIN {X 0,Y 587.846,Z 208.139,A -85,B 0,C 180,E1 -1551.935,E2 -1551.935} C_VEL
LIN {X 0,Y 587.793,Z 198.817,A -85,B 0,C 180,E1 -1553.235,E2 -1553.235} C_VEL
LIN {X 0,Y 587.334,Z 196.326,A -85,B 0,C 180,E1 -1553.628,E2 -1553.628} C_VEL
LIN {X 0,Y 587.35,Z 196.326,A -85,B 0,C 180,E1 -1556.274,E2 -1556.274} C_VEL
LIN {X 0,Y 587.33,Z 196.319,A -85,B 0,C 180,E1 -1559.13,E2 -1559.13} C_VEL
LIN {X 0,Y 587.325,Z 196.326,A -85,B 0,C 180,E1 -1561.832,E2 -1561.832} C_VEL
LIN {X 0,Y 587.333,Z 196.323,A -85,B 0,C 180,E1 -1564.345,E2 -1564.345} C_VEL
LIN {X 0,Y 587.326,Z 196.32,A -85,B 0,C 180,E1 -1566.743,E2 -1566.743} C_VEL
LIN {X 0,Y 587.321,Z 196.322,A -85,B 0,C 180,E1 -1569.355,E2 -1569.355} C_VEL
LIN {X 0,Y 587.302,Z 196.329,A -85,B 0,C 180,E1 -1572.104,E2 -1572.104} C_VEL
LIN {X 0,Y 587.28,Z 196.325,A -85,B 0,C 180,E1 -1574.907,E2 -1574.907} C_VEL
LIN {X 0,Y 587.314,Z 196.329,A -85,B 0,C 180,E1 -1577.924,E2 -1577.924} C_VEL
LIN {X 0,Y 587.313,Z 196.321,A -85,B 0,C 180,E1 -1580.638,E2 -1580.638} C_VEL
LIN {X 0,Y 587.312,Z 196.325,A -85,B 0,C 180,E1 -1583.288,E2 -1583.288} C_VEL
LIN {X 0,Y 587.331,Z 196.327,A -85,B 0,C 180,E1 -1585.778,E2 -1585.778} C_VEL
LIN {X 0,Y 587.32,Z 196.321,A -85,B 0,C 180,E1 -1588.23,E2 -1588.23} C_VEL
LIN {X 0,Y 587.329,Z 196.32,A -85,B 0,C 180,E1 -1590.858,E2 -1590.858} C_VEL
LIN {X 0,Y 587.311,Z 196.326,A -85,B 0,C 180,E1 -1593.814,E2 -1593.814} C_VEL
LIN {X 0,Y 587.324,Z 196.32,A -85,B 0,C 180,E1 -1596.741,E2 -1596.741} C_VEL
LIN {X 0,Y 587.299,Z 196.328,A -85,B 0,C 180,E1 -1599.694,E2 -1599.694} C_VEL
LIN {X 0,Y 587.287,Z 196.327,A -85,B 0,C 180,E1 -1601.872,E2 -1601.872} C_VEL
LIN {X 0,Y 587.287,Z 196.325,A -85,B 0,C 180,E1 -1604.024,E2 -1604.024} C_VEL
LIN {X 0,Y 587.295,Z 196.327,A -85,B 0,C 180,E1 -1606.858,E2 -1606.858} C_VEL
LIN {X 0,Y 587.349,Z 196.322,A -85,B 0,C 180,E1 -1608.963,E2 -1608.963} C_VEL
LIN {X 0,Y 587.314,Z 196.323,A -85,B 0,C 180,E1 -1611.744,E2 -1611.744} C_VEL
LIN {X 0,Y 587.273,Z 196.327,A -85,B 0,C 180,E1 -1613.817,E2 -1613.817} C_VEL
LIN {X 0,Y 587.255,Z 196.329,A -85,B 0,C 180,E1 -1615.882,E2 -1615.882} C_VEL
LIN {X 0,Y 587.3,Z 196.323,A -85,B 0,C 180,E1 -1617.943,E2 -1617.943} C_VEL
LIN {X 0,Y 587.347,Z 196.321,A -85,B 0,C 180,E1 -1620.686,E2 -1620.686} C_VEL
LIN {X 0,Y 587.291,Z 196.327,A -85,B 0,C 180,E1 -1623.43,E2 -1623.43} C_VEL
LIN {X 0,Y 587.309,Z 196.324,A -85,B 0,C 180,E1 -1625.494,E2 -1625.494} C_VEL
LIN {X 0,Y 587.309,Z 196.323,A -85,B 0,C 180,E1 -1628.256,E2 -1628.256} C_VEL
LIN {X 0,Y 587.366,Z 196.319,A -85,B 0,C 180,E1 -1631.177,E2 -1631.177} C_VEL
LIN {X 0,Y 587.316,Z 196.323,A -85,B 0,C 180,E1 -1634.268,E2 -1634.268} C_VEL
LIN {X 0,Y 587.304,Z 196.323,A -85,B 0,C 180,E1 -1637.408,E2 -1637.408} C_VEL
LIN {X 0,Y 587.282,Z 196.327,A -85,B 0,C 180,E1 -1638.344,E2 -1638.344} C_VEL
LIN {X 0,Y 586.635,Z 196.413,A -85,B 0,C 180,E1 -1638.916,E2 -1638.916} C_VEL
LIN {X 0,Y 583.797,Z 196.766,A -85,B 0,C 180,E1 -1639.845,E2 -1639.845} C_VEL
LIN {X 0,Y 581.38,Z 197.069,A -85,B 0,C 180,E1 -1640.592,E2 -1640.592} C_VEL
LIN {X 0,Y 580.33,Z 197.194,A -85,B 0,C 180,E1 -1641.168,E2 -1641.168} C_VEL
LIN {X 0,Y 580.238,Z 197.203,A -85,B 0,C 180,E1 -1641.363,E2 -1641.363} C_VEL
LIN {X 0,Y 580.248,Z 197.201,A -85,B 0,C 180,E1 -1643.559,E2 -1643.559} C_VEL
LIN {X 0,Y 580.275,Z 197.204,A -85,B 0,C 180,E1 -1646.345,E2 -1646.345} C_VEL
LIN {X 0,Y 580.273,Z 197.198,A -85,B 0,C 180,E1 -1649.317,E2 -1649.317} C_VEL
LIN {X 0,Y 580.263,Z 197.205,A -85,B 0,C 180,E1 -1652.203,E2 -1652.203} C_VEL
LIN {X 0,Y 580.259,Z 197.205,A -85,B 0,C 180,E1 -1654.699,E2 -1654.699} C_VEL
LIN {X 0,Y 580.258,Z 197.2,A -85,B 0,C 180,E1 -1657.272,E2 -1657.272} C_VEL
LIN {X 0,Y 580.261,Z 197.209,A -85,B 0,C 180,E1 -1660.276,E2 -1660.276} C_VEL
LIN {X 0,Y 580.261,Z 197.203,A -85,B 0,C 180,E1 -1662.708,E2 -1662.708} C_VEL
LIN {X 0,Y 580.24,Z 197.203,A -85,B 0,C 180,E1 -1665.613,E2 -1665.613} C_VEL
LIN {X 0,Y 580.284,Z 197.206,A -85,B 0,C 180,E1 -1668.238,E2 -1668.238} C_VEL
LIN {X 0,Y 580.257,Z 197.2,A -85,B 0,C 180,E1 -1670.97,E2 -1670.97} C_VEL
LIN {X 0,Y 580.268,Z 197.201,A -85,B 0,C 180,E1 -1673.602,E2 -1673.602} C_VEL
LIN {X 0,Y 580.284,Z 197.198,A -85,B 0,C 180,E1 -1676.687,E2 -1676.687} C_VEL
LIN {X 0,Y 580.284,Z 197.198,A -85,B 0,C 180,E1 -1679.429,E2 -1679.429} C_VEL
LIN {X 0,Y 580.283,Z 197.204,A -85,B 0,C 180,E1 -1682.145,E2 -1682.145} C_VEL
LIN {X 0,Y 580.31,Z 197.195,A -85,B 0,C 180,E1 -1685.273,E2 -1685.273} C_VEL
LIN {X 0,Y 580.259,Z 197.208,A -85,B 0,C 180,E1 -1687.951,E2 -1687.951} C_VEL
LIN {X 0,Y 580.28,Z 197.197,A -85,B 0,C 180,E1 -1690.916,E2 -1690.916} C_VEL
LIN {X 0,Y 580.253,Z 197.209,A -85,B 0,C 180,E1 -1693.828,E2 -1693.828} C_VEL
LIN {X 0,Y 580.31,Z 197.199,A -85,B 0,C 180,E1 -1695.985,E2 -1695.985} C_VEL
LIN {X 0,Y 580.305,Z 197.195,A -85,B 0,C 180,E1 -1698.829,E2 -1698.829} C_VEL
LIN {X 0,Y 580.325,Z 197.202,A -85,B 0,C 180,E1 -1701.646,E2 -1701.646} C_VEL
LIN {X 0,Y 580.314,Z 197.383,A -85,B 0,C 180,E1 -1702.74,E2 -1702.74} C_VEL
LIN {X 0,Y 580.387,Z 206.53,A -85,B 0,C 180,E1 -1704.443,E2 -1704.443} C_VEL
LIN {X 0,Y 580.338,Z 221.677,A -85,B 0,C 180,E1 -1707.225,E2 -1707.225} C_VEL
LIN {X 0,Y 580.338,Z 222.628,A -85,B 0,C 180,E1 -1707.399,E2 -1707.399} C_VEL
LIN {X 0,Y 580.942,Z 228.202,A -85,B 0,C 180,E1 -1707.488,E2 -1707.488} C_VEL
LIN {X 0,Y 580.776,Z 329.657,A -85,B 0,C 180,E1 -1708.766,E2 -1708.766} C_VEL
LIN {X 0,Y 580.733,Z 343.223,A -85,B 0,C 180,E1 -1709.091,E2 -1709.091} C_VEL
LIN {X 0,Y 580.631,Z 355.481,A -85,B 0,C 180,E1 -1709.525,E2 -1709.525} C_VEL
LIN {X 0,Y 580.548,Z 367.25,A -85,B 0,C 180,E1 -1710.088,E2 -1710.088} C_VEL
LIN {X 0,Y 580.366,Z 378.581,A -85,B 0,C 180,E1 -1710.782,E2 -1710.782} C_VEL
LIN {X 0,Y 580.361,Z 388.773,A -85,B 0,C 180,E1 -1711.562,E2 -1711.562} C_VEL
LIN {X 0,Y 580.24,Z 398.031,A -85,B 0,C 180,E1 -1712.431,E2 -1712.431} C_VEL
LIN {X 0,Y 580.169,Z 407,A -85,B 0,C 180,E1 -1713.473,E2 -1713.473} C_VEL
LIN {X 0,Y 580.154,Z 414.253,A -85,B 0,C 180,E1 -1714.517,E2 -1714.517} C_VEL
LIN {X 0,Y 580.132,Z 420.089,A -85,B 0,C 180,E1 -1715.562,E2 -1715.562} C_VEL
LIN {X 0,Y 580.11,Z 424.546,A -85,B 0,C 180,E1 -1716.571,E2 -1716.571} C_VEL
LIN {X 0,Y 580.071,Z 428.224,A -85,B 0,C 180,E1 -1717.659,E2 -1717.659} C_VEL
LIN {X 0,Y 580.062,Z 430.014,A -85,B 0,C 180,E1 -1718.36,E2 -1718.36} C_VEL
LIN {X 0,Y 580.057,Z 432.309,A -85,B 0,C 180,E1 -1719.766,E2 -1719.766} C_VEL
LIN {X 0,Y 580.074,Z 432.998,A -85,B 0,C 180,E1 -1721.075,E2 -1721.075} C_VEL
LIN {X 0,Y 580.054,Z 432.686,A -85,B 0,C 180,E1 -1721.887,E2 -1721.887} C_VEL
LIN {X 0,Y 580.051,Z 431.997,A -85,B 0,C 180,E1 -1722.597,E2 -1722.597} C_VEL
LIN {X 0,Y 580.066,Z 430.883,A -85,B 0,C 180,E1 -1723.309,E2 -1723.309} C_VEL
LIN {X 0,Y 580.087,Z 428.726,A -85,B 0,C 180,E1 -1724.248,E2 -1724.248} C_VEL
LIN {X 0,Y 580.095,Z 424.793,A -85,B 0,C 180,E1 -1725.458,E2 -1725.458} C_VEL
LIN {X 0,Y 580.099,Z 420.148,A -85,B 0,C 180,E1 -1726.517,E2 -1726.517} C_VEL
LIN {X 0,Y 580.139,Z 413.896,A -85,B 0,C 180,E1 -1727.629,E2 -1727.629} C_VEL
LIN {X 0,Y 580.187,Z 406.172,A -85,B 0,C 180,E1 -1728.723,E2 -1728.723} C_VEL
LIN {X 0,Y 580.295,Z 398.224,A -85,B 0,C 180,E1 -1729.638,E2 -1729.638} C_VEL
LIN {X 0,Y 580.342,Z 388.392,A -85,B 0,C 180,E1 -1730.56,E2 -1730.56} C_VEL
LIN {X 0,Y 580.413,Z 377.331,A -85,B 0,C 180,E1 -1731.393,E2 -1731.393} C_VEL
LIN {X 0,Y 580.535,Z 366.55,A -85,B 0,C 180,E1 -1732.041,E2 -1732.041} C_VEL
LIN {X 0,Y 580.615,Z 354.613,A -85,B 0,C 180,E1 -1732.6,E2 -1732.6} C_VEL
LIN {X 0,Y 580.695,Z 341.414,A -85,B 0,C 180,E1 -1733.052,E2 -1733.052} C_VEL
LIN {X 0,Y 580.753,Z 328.18,A -85,B 0,C 180,E1 -1733.352,E2 -1733.352} C_VEL
LIN {X 0,Y 580.881,Z 226.257,A -85,B 0,C 180,E1 -1734.628,E2 -1734.628} C_VEL
LIN {X 0,Y 580.257,Z 222.6,A -85,B 0,C 180,E1 -1734.698,E2 -1734.698} C_VEL
LIN {X 0,Y 580.352,Z 207.889,A -85,B 0,C 180,E1 -1737.397,E2 -1737.397} C_VEL
LIN {X 0,Y 580.335,Z 197.194,A -85,B 0,C 180,E1 -1739.399,E2 -1739.399} C_VEL
LIN {X 0,Y 580.296,Z 197.202,A -85,B 0,C 180,E1 -1742.199,E2 -1742.199} C_VEL
LIN {X 0,Y 580.293,Z 197.201,A -85,B 0,C 180,E1 -1744.694,E2 -1744.694} C_VEL
LIN {X 0,Y 580.291,Z 197.197,A -85,B 0,C 180,E1 -1747.266,E2 -1747.266} C_VEL
LIN {X 0,Y 580.295,Z 197.205,A -85,B 0,C 180,E1 -1750.27,E2 -1750.27} C_VEL
LIN {X 0,Y 580.268,Z 197.202,A -85,B 0,C 180,E1 -1752.704,E2 -1752.704} C_VEL
LIN {X 0,Y 580.257,Z 197.202,A -85,B 0,C 180,E1 -1755.607,E2 -1755.607} C_VEL
LIN {X 0,Y 580.296,Z 197.203,A -85,B 0,C 180,E1 -1758.232,E2 -1758.232} C_VEL
LIN {X 0,Y 580.272,Z 197.198,A -85,B 0,C 180,E1 -1760.964,E2 -1760.964} C_VEL
LIN {X 0,Y 580.275,Z 197.202,A -85,B 0,C 180,E1 -1763.597,E2 -1763.597} C_VEL
LIN {X 0,Y 580.3,Z 197.201,A -85,B 0,C 180,E1 -1766.144,E2 -1766.144} C_VEL
LIN {X 0,Y 580.268,Z 197.199,A -85,B 0,C 180,E1 -1768.614,E2 -1768.614} C_VEL
LIN {X 0,Y 580.276,Z 197.198,A -85,B 0,C 180,E1 -1771.023,E2 -1771.023} C_VEL
LIN {X 0,Y 580.298,Z 197.203,A -85,B 0,C 180,E1 -1773.656,E2 -1773.656} C_VEL
LIN {X 0,Y 580.274,Z 197.198,A -85,B 0,C 180,E1 -1776.442,E2 -1776.442} C_VEL
LIN {X 0,Y 580.265,Z 197.206,A -85,B 0,C 180,E1 -1779.437,E2 -1779.437} C_VEL
LIN {X 0,Y 580.261,Z 197.209,A -85,B 0,C 180,E1 -1781.645,E2 -1781.645} C_VEL
LIN {X 0,Y 580.263,Z 197.204,A -85,B 0,C 180,E1 -1783.825,E2 -1783.825} C_VEL
LIN {X 0,Y 580.299,Z 197.198,A -85,B 0,C 180,E1 -1785.982,E2 -1785.982} C_VEL
LIN {X 0,Y 580.313,Z 197.194,A -85,B 0,C 180,E1 -1788.827,E2 -1788.827} C_VEL
LIN {X 0,Y 580.3,Z 197.2,A -85,B 0,C 180,E1 -1791.643,E2 -1791.643} C_VEL
LIN {X 0,Y 580.251,Z 197.204,A -85,B 0,C 180,E1 -1793.742,E2 -1793.742} C_VEL
LIN {X 0,Y 580.231,Z 197.205,A -85,B 0,C 180,E1 -1795.832,E2 -1795.832} C_VEL
LIN {X 0,Y 580.291,Z 197.196,A -85,B 0,C 180,E1 -1797.918,E2 -1797.918} C_VEL
LIN {X 0,Y 580.301,Z 197.195,A -85,B 0,C 180,E1 -1800,E2 -1800} C_VEL
LIN {X 0,Y 580.309,Z 197.197,A -85,B 0,C 180,E1 -1802.777,E2 -1802.777} C_VEL
LIN {X 0,Y 580.29,Z 197.199,A -85,B 0,C 180,E1 -1805.56,E2 -1805.56} C_VEL
LIN {X 0,Y 580.265,Z 197.199,A -85,B 0,C 180,E1 -1808.357,E2 -1808.357} C_VEL
LIN {X 0,Y 580.325,Z 197.197,A -85,B 0,C 180,E1 -1811.224,E2 -1811.224} C_VEL
LIN {X 0,Y 580.268,Z 197.2,A -85,B 0,C 180,E1 -1814.336,E2 -1814.336} C_VEL
LIN {X 0,Y 580.275,Z 197.207,A -85,B 0,C 180,E1 -1816.915,E2 -1816.915} C_VEL
LIN {X 0,Y 580.249,Z 197.201,A -85,B 0,C 180,E1 -1819.824,E2 -1819.824} C_VEL
LIN {X 0,Y 580.231,Z 197.204,A -85,B 0,C 180,E1 -1822.054,E2 -1822.054} C_VEL
LIN {X 0,Y 580.263,Z 197.202,A -85,B 0,C 180,E1 -1825.082,E2 -1825.082} C_VEL
LIN {X 0,Y 580.253,Z 197.204,A -85,B 0,C 180,E1 -1828.188,E2 -1828.188} C_VEL
LIN {X 0,Y 580.244,Z 197.21,A -85,B 0,C 180,E1 -1830.695,E2 -1830.695} C_VEL
LIN {X 0,Y 580.253,Z 197.2,A -85,B 0,C 180,E1 -1833.315,E2 -1833.315} C_VEL
LIN {X 0,Y 580.218,Z 197.206,A -85,B 0,C 180,E1 -1835.758,E2 -1835.758} C_VEL
LIN {X 0,Y 580.262,Z 197.204,A -85,B 0,C 180,E1 -1838.149,E2 -1838.149} C_VEL
LIN {X 0,Y 580.276,Z 197.2,A -85,B 0,C 180,E1 -1840.846,E2 -1840.846} C_VEL
LIN {X 0,Y 580.252,Z 197.202,A -85,B 0,C 180,E1 -1843.661,E2 -1843.661} C_VEL
LIN {X 0,Y 580.248,Z 197.205,A -85,B 0,C 180,E1 -1846.613,E2 -1846.613} C_VEL
LIN {X 0,Y 580.279,Z 197.197,A -85,B 0,C 180,E1 -1849.158,E2 -1849.158} C_VEL
LIN {X 0,Y 580.274,Z 197.205,A -85,B 0,C 180,E1 -1851.929,E2 -1851.929} C_VEL
LIN {X 0,Y 580.271,Z 197.202,A -85,B 0,C 180,E1 -1854.456,E2 -1854.456} C_VEL
LIN {X 0,Y 580.28,Z 197.197,A -85,B 0,C 180,E1 -1856.977,E2 -1856.977} C_VEL
LIN {X 0,Y 580.287,Z 197.199,A -85,B 0,C 180,E1 -1859.426,E2 -1859.426} C_VEL
LIN {X 0,Y 580.253,Z 197.207,A -85,B 0,C 180,E1 -1862.15,E2 -1862.15} C_VEL
LIN {X 0,Y 580.301,Z 197.197,A -85,B 0,C 180,E1 -1864.921,E2 -1864.921} C_VEL
LIN {X 0,Y 580.312,Z 197.39,A -85,B 0,C 180,E1 -1866.302,E2 -1866.302} C_VEL
LIN {X 0,Y 580.948,Z 201.949,A -85,B 0,C 180,E1 -1866.956,E2 -1866.956} C_VEL
LIN {X 0,Y 580.837,Z 221.414,A -85,B 0,C 180,E1 -1869.644,E2 -1869.644} C_VEL
LIN {X 0,Y 580.587,Z 242.819,A -85,B 0,C 180,E1 -1872.585,E2 -1872.585} C_VEL
LIN {X 0,Y 580.465,Z 262.628,A -85,B 0,C 180,E1 -1875.271,E2 -1875.271} C_VEL
LIN {X 0,Y 580.413,Z 270.522,A -85,B 0,C 180,E1 -1876.331,E2 -1876.331} C_VEL
LIN {X 0,Y 580.96,Z 276.509,A -85,B 0,C 180,E1 -1876.422,E2 -1876.422} C_VEL
LIN {X 0,Y 580.802,Z 378.94,A -85,B 0,C 180,E1 -1877.708,E2 -1877.708} C_VEL
LIN {X 0,Y 580.74,Z 392.214,A -85,B 0,C 180,E1 -1878.017,E2 -1878.017} C_VEL
LIN {X 0,Y 580.656,Z 405.143,A -85,B 0,C 180,E1 -1878.466,E2 -1878.466} C_VEL
LIN {X 0,Y 580.553,Z 416.624,A -85,B 0,C 180,E1 -1879.008,E2 -1879.008} C_VEL
LIN {X 0,Y 580.445,Z 428.197,A -85,B 0,C 180,E1 -1879.712,E2 -1879.712} C_VEL
LIN {X 0,Y 580.345,Z 438.596,A -85,B 0,C 180,E1 -1880.502,E2 -1880.502} C_VEL
LIN {X 0,Y 580.272,Z 447.108,A -85,B 0,C 180,E1 -1881.292,E2 -1881.292} C_VEL
LIN {X 0,Y 580.222,Z 454.956,A -85,B 0,C 180,E1 -1882.168,E2 -1882.168} C_VEL
LIN {X 0,Y 580.154,Z 462.648,A -85,B 0,C 180,E1 -1883.221,E2 -1883.221} C_VEL
LIN {X 0,Y 580.139,Z 469.676,A -85,B 0,C 180,E1 -1884.438,E2 -1884.438} C_VEL
LIN {X 0,Y 580.108,Z 474.368,A -85,B 0,C 180,E1 -1885.483,E2 -1885.483} C_VEL
LIN {X 0,Y 580.123,Z 477.954,A -85,B 0,C 180,E1 -1886.526,E2 -1886.526} C_VEL
LIN {X 0,Y 580.043,Z 479.806,A -85,B 0,C 180,E1 -1887.221,E2 -1887.221} C_VEL
LIN {X 0,Y 580.04,Z 481.197,A -85,B 0,C 180,E1 -1887.916,E2 -1887.916} C_VEL
LIN {X 0,Y 580.04,Z 482.784,A -85,B 0,C 180,E1 -1889.305,E2 -1889.305} C_VEL
LIN {X 0,Y 580.037,Z 483,A -85,B 0,C 180,E1 -1889.999,E2 -1889.999} C_VEL
LIN {X 0,Y 580.047,Z 482.188,A -85,B 0,C 180,E1 -1891.387,E2 -1891.387} C_VEL
LIN {X 0,Y 580.04,Z 481.202,A -85,B 0,C 180,E1 -1892.082,E2 -1892.082} C_VEL
LIN {X 0,Y 580.043,Z 479.814,A -85,B 0,C 180,E1 -1892.776,E2 -1892.776} C_VEL
LIN {X 0,Y 580.109,Z 476.901,A -85,B 0,C 180,E1 -1893.819,E2 -1893.819} C_VEL
LIN {X 0,Y 580.053,Z 472.956,A -85,B 0,C 180,E1 -1894.863,E2 -1894.863} C_VEL
LIN {X 0,Y 580.166,Z 467.877,A -85,B 0,C 180,E1 -1895.908,E2 -1895.908} C_VEL
LIN {X 0,Y 580.183,Z 460.252,A -85,B 0,C 180,E1 -1897.13,E2 -1897.13} C_VEL
LIN {X 0,Y 580.249,Z 452.009,A -85,B 0,C 180,E1 -1898.18,E2 -1898.18} C_VEL
LIN {X 0,Y 580.307,Z 443.562,A -85,B 0,C 180,E1 -1899.056,E2 -1899.056} C_VEL
LIN {X 0,Y 580.424,Z 433.128,A -85,B 0,C 180,E1 -1899.933,E2 -1899.933} C_VEL
LIN {X 0,Y 580.491,Z 422.793,A -85,B 0,C 180,E1 -1900.637,E2 -1900.637} C_VEL
LIN {X 0,Y 580.592,Z 411.286,A -85,B 0,C 180,E1 -1901.262,E2 -1901.262} C_VEL
LIN {X 0,Y 580.676,Z 398.545,A -85,B 0,C 180,E1 -1901.782,E2 -1901.782} C_VEL
LIN {X 0,Y 580.78,Z 385.538,A -85,B 0,C 180,E1 -1902.157,E2 -1902.157} C_VEL
LIN {X 0,Y 580.81,Z 373.268,A -85,B 0,C 180,E1 -1902.378,E2 -1902.378} C_VEL
LIN {X 0,Y 580.802,Z 273.372,A -85,B 0,C 180,E1 -1903.62,E2 -1903.62} C_VEL
LIN {X 0,Y 580.406,Z 270.459,A -85,B 0,C 180,E1 -1903.677,E2 -1903.677} C_VEL
LIN {X 0,Y 580.594,Z 248.024,A -85,B 0,C 180,E1 -1906.705,E2 -1906.705} C_VEL
LIN {X 0,Y 580.776,Z 226.609,A -85,B 0,C 180,E1 -1909.638,E2 -1909.638} C_VEL
LIN {X 0,Y 580.938,Z 206.666,A -85,B 0,C 180,E1 -1912.397,E2 -1912.397} C_VEL
LIN {X 0,Y 580.864,Z 200.233,A -85,B 0,C 180,E1 -1913.288,E2 -1913.288} C_VEL
LIN {X 0,Y 580.285,Z 197.205,A -85,B 0,C 180,E1 -1913.743,E2 -1913.743} C_VEL
LIN {X 0,Y 580.292,Z 197.2,A -85,B 0,C 180,E1 -1916.618,E2 -1916.618} C_VEL
LIN {X 0,Y 580.286,Z 197.197,A -85,B 0,C 180,E1 -1919.306,E2 -1919.306} C_VEL
LIN {X 0,Y 580.278,Z 197.205,A -85,B 0,C 180,E1 -1922.197,E2 -1922.197} C_VEL
LIN {X 0,Y 580.277,Z 197.198,A -85,B 0,C 180,E1 -1924.692,E2 -1924.692} C_VEL
LIN {X 0,Y 580.275,Z 197.199,A -85,B 0,C 180,E1 -1927.264,E2 -1927.264} C_VEL
LIN {X 0,Y 580.271,Z 197.202,A -85,B 0,C 180,E1 -1930.268,E2 -1930.268} C_VEL
LIN {X 0,Y 580.248,Z 197.201,A -85,B 0,C 180,E1 -1932.702,E2 -1932.702} C_VEL
LIN {X 0,Y 580.238,Z 197.209,A -85,B 0,C 180,E1 -1935.605,E2 -1935.605} C_VEL
LIN {X 0,Y 580.282,Z 197.2,A -85,B 0,C 180,E1 -1938.231,E2 -1938.231} C_VEL
LIN {X 0,Y 580.254,Z 197.201,A -85,B 0,C 180,E1 -1940.963,E2 -1940.963} C_VEL
LIN {X 0,Y 580.255,Z 197.209,A -85,B 0,C 180,E1 -1943.595,E2 -1943.595} C_VEL
LIN {X 0,Y 580.284,Z 197.199,A -85,B 0,C 180,E1 -1946.143,E2 -1946.143} C_VEL
LIN {X 0,Y 580.25,Z 197.201,A -85,B 0,C 180,E1 -1948.613,E2 -1948.613} C_VEL
LIN {X 0,Y 580.273,Z 197.2,A -85,B 0,C 180,E1 -1951.023,E2 -1951.023} C_VEL
LIN {X 0,Y 580.277,Z 197.205,A -85,B 0,C 180,E1 -1953.655,E2 -1953.655} C_VEL
LIN {X 0,Y 580.255,Z 197.2,A -85,B 0,C 180,E1 -1956.441,E2 -1956.441} C_VEL
LIN {X 0,Y 580.279,Z 197.199,A -85,B 0,C 180,E1 -1958.822,E2 -1958.822} C_VEL
LIN {X 0,Y 580.243,Z 197.207,A -85,B 0,C 180,E1 -1961.644,E2 -1961.644} C_VEL
LIN {X 0,Y 580.244,Z 197.204,A -85,B 0,C 180,E1 -1963.825,E2 -1963.825} C_VEL
LIN {X 0,Y 580.246,Z 197.203,A -85,B 0,C 180,E1 -1966.695,E2 -1966.695} C_VEL
LIN {X 0,Y 580.269,Z 197.203,A -85,B 0,C 180,E1 -1969.533,E2 -1969.533} C_VEL
LIN {X 0,Y 580.28,Z 197.197,A -85,B 0,C 180,E1 -1972.344,E2 -1972.344} C_VEL
LIN {X 0,Y 580.295,Z 197.206,A -85,B 0,C 180,E1 -1975.137,E2 -1975.137} C_VEL
LIN {X 0,Y 580.271,Z 197.198,A -85,B 0,C 180,E1 -1977.918,E2 -1977.918} C_VEL
LIN {X 0,Y 580.316,Z 197.197,A -85,B 0,C 180,E1 -1980.694,E2 -1980.694} C_VEL
LIN {X 0,Y 580.241,Z 197.205,A -85,B 0,C 180,E1 -1983.472,E2 -1983.472} C_VEL
LIN {X 0,Y 580.272,Z 197.2,A -85,B 0,C 180,E1 -1985.56,E2 -1985.56} C_VEL
LIN {X 0,Y 580.274,Z 197.2,A -85,B 0,C 180,E1 -1988.357,E2 -1988.357} C_VEL
LIN {X 0,Y 580.319,Z 197.196,A -85,B 0,C 180,E1 -1991.234,E2 -1991.234} C_VEL
LIN {X 0,Y 580.263,Z 197.202,A -85,B 0,C 180,E1 -1994.345,E2 -1994.345} C_VEL
LIN {X 0,Y 580.283,Z 197.204,A -85,B 0,C 180,E1 -1996.927,E2 -1996.927} C_VEL
LIN {X 0,Y 580.259,Z 197.2,A -85,B 0,C 180,E1 -1999.824,E2 -1999.824} C_VEL
LIN {X 0,Y 580.238,Z 197.203,A -85,B 0,C 180,E1 -2001.363,E2 -2001.363} C_VEL
LIN {X 0,Y 579.55,Z 197.289,A -85,B 0,C 180,E1 -2001.943,E2 -2001.943} C_VEL
LIN {X 0,Y 576.676,Z 197.652,A -85,B 0,C 180,E1 -2002.883,E2 -2002.883} C_VEL
LIN {X 0,Y 574.275,Z 197.948,A -85,B 0,C 180,E1 -2003.64,E2 -2003.64} C_VEL
LIN {X 0,Y 573.27,Z 198.074,A -85,B 0,C 180,E1 -2004.224,E2 -2004.224} C_VEL
LIN {X 0,Y 573.201,Z 198.085,A -85,B 0,C 180,E1 -2004.421,E2 -2004.421} C_VEL
LIN {X 0,Y 573.216,Z 198.081,A -85,B 0,C 180,E1 -2006.978,E2 -2006.978} C_VEL
LIN {X 0,Y 573.215,Z 198.077,A -85,B 0,C 180,E1 -2009.495,E2 -2009.495} C_VEL
LIN {X 0,Y 573.214,Z 198.084,A -85,B 0,C 180,E1 -2012.648,E2 -2012.648} C_VEL
LIN {X 0,Y 573.225,Z 198.076,A -85,B 0,C 180,E1 -2015.187,E2 -2015.187} C_VEL
LIN {X 0,Y 573.195,Z 198.081,A -85,B 0,C 180,E1 -2017.811,E2 -2017.811} C_VEL
LIN {X 0,Y 573.23,Z 198.082,A -85,B 0,C 180,E1 -2020.532,E2 -2020.532} C_VEL
LIN {X 0,Y 573.211,Z 198.078,A -85,B 0,C 180,E1 -2023.362,E2 -2023.362} C_VEL
LIN {X 0,Y 573.219,Z 198.085,A -85,B 0,C 180,E1 -2026.334,E2 -2026.334} C_VEL
LIN {X 0,Y 573.245,Z 198.074,A -85,B 0,C 180,E1 -2029.481,E2 -2029.481} C_VEL
LIN {X 0,Y 573.21,Z 198.087,A -85,B 0,C 180,E1 -2032.196,E2 -2032.196} C_VEL
LIN {X 0,Y 573.232,Z 198.076,A -85,B 0,C 180,E1 -2034.819,E2 -2034.819} C_VEL
LIN {X 0,Y 573.233,Z 198.076,A -85,B 0,C 180,E1 -2037.359,E2 -2037.359} C_VEL
LIN {X 0,Y 573.233,Z 198.077,A -85,B 0,C 180,E1 -2040.515,E2 -2040.515} C_VEL
LIN {X 0,Y 573.205,Z 198.078,A -85,B 0,C 180,E1 -2043.026,E2 -2043.026} C_VEL
LIN {X 0,Y 573.264,Z 198.073,A -85,B 0,C 180,E1 -2045.37,E2 -2045.37} C_VEL
LIN {X 0,Y 573.219,Z 198.078,A -85,B 0,C 180,E1 -2048.423,E2 -2048.423} C_VEL
LIN {X 0,Y 573.263,Z 198.071,A -85,B 0,C 180,E1 -2050.734,E2 -2050.734} C_VEL
LIN {X 0,Y 573.226,Z 198.084,A -85,B 0,C 180,E1 -2053.624,E2 -2053.624} C_VEL
LIN {X 0,Y 573.255,Z 198.081,A -85,B 0,C 180,E1 -2055.809,E2 -2055.809} C_VEL
LIN {X 0,Y 573.263,Z 198.072,A -85,B 0,C 180,E1 -2058.748,E2 -2058.748} C_VEL
LIN {X 0,Y 573.28,Z 198.079,A -85,B 0,C 180,E1 -2061.543,E2 -2061.543} C_VEL
LIN {X 0,Y 573.248,Z 198.137,A -85,B 0,C 180,E1 -2062.65,E2 -2062.65} C_VEL
LIN {X 0,Y 573.399,Z 205.397,A -85,B 0,C 180,E1 -2064.022,E2 -2064.022} C_VEL
LIN {X 0,Y 573.247,Z 218.636,A -85,B 0,C 180,E1 -2066.487,E2 -2066.487} C_VEL
LIN {X 0,Y 573.314,Z 222.72,A -85,B 0,C 180,E1 -2067.235,E2 -2067.235} C_VEL
LIN {X 0,Y 574.044,Z 228.537,A -85,B 0,C 180,E1 -2067.326,E2 -2067.326} C_VEL
LIN {X 0,Y 573.85,Z 328.743,A -85,B 0,C 180,E1 -2068.598,E2 -2068.598} C_VEL
LIN {X 0,Y 573.798,Z 341.871,A -85,B 0,C 180,E1 -2068.905,E2 -2068.905} C_VEL
LIN {X 0,Y 573.681,Z 354.49,A -85,B 0,C 180,E1 -2069.343,E2 -2069.343} C_VEL
LIN {X 0,Y 573.557,Z 366.555,A -85,B 0,C 180,E1 -2069.914,E2 -2069.914} C_VEL
LIN {X 0,Y 573.361,Z 378.012,A -85,B 0,C 180,E1 -2070.616,E2 -2070.616} C_VEL
LIN {X 0,Y 573.347,Z 388.306,A -85,B 0,C 180,E1 -2071.406,E2 -2071.406} C_VEL
LIN {X 0,Y 573.201,Z 397.663,A -85,B 0,C 180,E1 -2072.285,E2 -2072.285} C_VEL
LIN {X 0,Y 573.115,Z 406.698,A -85,B 0,C 180,E1 -2073.34,E2 -2073.34} C_VEL
LIN {X 0,Y 573.072,Z 414.006,A -85,B 0,C 180,E1 -2074.397,E2 -2074.397} C_VEL
LIN {X 0,Y 573.054,Z 420.742,A -85,B 0,C 180,E1 -2075.631,E2 -2075.631} C_VEL
LIN {X 0,Y 573.032,Z 424.755,A -85,B 0,C 180,E1 -2076.568,E2 -2076.568} C_VEL
LIN {X 0,Y 572.981,Z 428.606,A -85,B 0,C 180,E1 -2077.755,E2 -2077.755} C_VEL
LIN {X 0,Y 572.952,Z 430.297,A -85,B 0,C 180,E1 -2078.465,E2 -2078.465} C_VEL
LIN {X 0,Y 572.974,Z 432.462,A -85,B 0,C 180,E1 -2079.888,E2 -2079.888} C_VEL
LIN {X 0,Y 572.986,Z 432.991,A -85,B 0,C 180,E1 -2081.113,E2 -2081.113} C_VEL
LIN {X 0,Y 572.948,Z 432.59,A -85,B 0,C 180,E1 -2082.036,E2 -2082.036} C_VEL
LIN {X 0,Y 572.948,Z 431.824,A -85,B 0,C 180,E1 -2082.756,E2 -2082.756} C_VEL
LIN {X 0,Y 572.976,Z 430.599,A -85,B 0,C 180,E1 -2083.477,E2 -2083.477} C_VEL
LIN {X 0,Y 572.996,Z 428.667,A -85,B 0,C 180,E1 -2084.311,E2 -2084.311} C_VEL
LIN {X 0,Y 572.993,Z 425.591,A -85,B 0,C 180,E1 -2085.29,E2 -2085.29} C_VEL
LIN {X 0,Y 573.007,Z 421.081,A -85,B 0,C 180,E1 -2086.385,E2 -2086.385} C_VEL
LIN {X 0,Y 573.109,Z 415.283,A -85,B 0,C 180,E1 -2087.484,E2 -2087.484} C_VEL
LIN {X 0,Y 573.122,Z 407.906,A -85,B 0,C 180,E1 -2088.592,E2 -2088.592} C_VEL
LIN {X 0,Y 573.246,Z 398.602,A -85,B 0,C 180,E1 -2089.703,E2 -2089.703} C_VEL
LIN {X 0,Y 573.323,Z 388.893,A -85,B 0,C 180,E1 -2090.635,E2 -2090.635} C_VEL
LIN {X 0,Y 573.409,Z 377.799,A -85,B 0,C 180,E1 -2091.488,E2 -2091.488} C_VEL
LIN {X 0,Y 573.537,Z 367.293,A -85,B 0,C 180,E1 -2092.135,E2 -2092.135} C_VEL
LIN {X 0,Y 573.639,Z 355.667,A -85,B 0,C 180,E1 -2092.7,E2 -2092.7} C_VEL
LIN {X 0,Y 573.741,Z 342.632,A -85,B 0,C 180,E1 -2093.164,E2 -2093.164} C_VEL
LIN {X 0,Y 573.826,Z 329.523,A -85,B 0,C 180,E1 -2093.477,E2 -2093.477} C_VEL
LIN {X 0,Y 573.946,Z 226.911,A -85,B 0,C 180,E1 -2094.787,E2 -2094.787} C_VEL
LIN {X 0,Y 573.223,Z 222.609,A -85,B 0,C 180,E1 -2094.868,E2 -2094.868} C_VEL
LIN {X 0,Y 573.355,Z 208.106,A -85,B 0,C 180,E1 -2097.562,E2 -2097.562} C_VEL
LIN {X 0,Y 573.285,Z 198.073,A -85,B 0,C 180,E1 -2099.471,E2 -2099.471} C_VEL
LIN {X 0,Y 573.25,Z 198.08,A -85,B 0,C 180,E1 -2102.643,E2 -2102.643} C_VEL
LIN {X 0,Y 573.26,Z 198.073,A -85,B 0,C 180,E1 -2105.182,E2 -2105.182} C_VEL
LIN {X 0,Y 573.228,Z 198.079,A -85,B 0,C 180,E1 -2107.805,E2 -2107.805} C_VEL
LIN {X 0,Y 573.258,Z 198.078,A -85,B 0,C 180,E1 -2110.526,E2 -2110.526} C_VEL
LIN {X 0,Y 573.238,Z 198.077,A -85,B 0,C 180,E1 -2113.668,E2 -2113.668} C_VEL
LIN {X 0,Y 573.235,Z 198.078,A -85,B 0,C 180,E1 -2116.64,E2 -2116.64} C_VEL
LIN {X 0,Y 573.255,Z 198.074,A -85,B 0,C 180,E1 -2119.475,E2 -2119.475} C_VEL
LIN {X 0,Y 573.217,Z 198.084,A -85,B 0,C 180,E1 -2122.191,E2 -2122.191} C_VEL
LIN {X 0,Y 573.246,Z 198.074,A -85,B 0,C 180,E1 -2124.815,E2 -2124.815} C_VEL
LIN {X 0,Y 573.235,Z 198.077,A -85,B 0,C 180,E1 -2127.353,E2 -2127.353} C_VEL
LIN {X 0,Y 573.232,Z 198.084,A -85,B 0,C 180,E1 -2129.823,E2 -2129.823} C_VEL
LIN {X 0,Y 573.262,Z 198.074,A -85,B 0,C 180,E1 -2132.233,E2 -2132.233} C_VEL
LIN {X 0,Y 573.238,Z 198.076,A -85,B 0,C 180,E1 -2135.12,E2 -2135.12} C_VEL
LIN {X 0,Y 573.23,Z 198.085,A -85,B 0,C 180,E1 -2137.662,E2 -2137.662} C_VEL
LIN {X 0,Y 573.243,Z 198.073,A -85,B 0,C 180,E1 -2140.669,E2 -2140.669} C_VEL
LIN {X 0,Y 573.239,Z 198.082,A -85,B 0,C 180,E1 -2143.621,E2 -2143.621} C_VEL
LIN {X 0,Y 573.21,Z 198.078,A -85,B 0,C 180,E1 -2146.529,E2 -2146.529} C_VEL
LIN {X 0,Y 573.247,Z 198.082,A -85,B 0,C 180,E1 -2149.403,E2 -2149.403} C_VEL
LIN {X 0,Y 573.252,Z 198.073,A -85,B 0,C 180,E1 -2152.249,E2 -2152.249} C_VEL
LIN {X 0,Y 573.256,Z 198.072,A -85,B 0,C 180,E1 -2154.371,E2 -2154.371} C_VEL
LIN {X 0,Y 573.282,Z 198.078,A -85,B 0,C 180,E1 -2157.189,E2 -2157.189} C_VEL
LIN {X 0,Y 573.271,Z 198.071,A -85,B 0,C 180,E1 -2160,E2 -2160} C_VEL
LIN {X 0,Y 573.275,Z 198.074,A -85,B 0,C 180,E1 -2162.811,E2 -2162.811} C_VEL
LIN {X 0,Y 573.255,Z 198.074,A -85,B 0,C 180,E1 -2165.628,E2 -2165.628} C_VEL
LIN {X 0,Y 573.231,Z 198.075,A -85,B 0,C 180,E1 -2167.751,E2 -2167.751} C_VEL
LIN {X 0,Y 573.255,Z 198.076,A -85,B 0,C 180,E1 -2170.597,E2 -2170.597} C_VEL
LIN {X 0,Y 573.189,Z 198.082,A -85,B 0,C 180,E1 -2173.472,E2 -2173.472} C_VEL
LIN {X 0,Y 573.194,Z 198.08,A -85,B 0,C 180,E1 -2175.649,E2 -2175.649} C_VEL
LIN {X 0,Y 573.201,Z 198.079,A -85,B 0,C 180,E1 -2177.85,E2 -2177.85} C_VEL
LIN {X 0,Y 573.207,Z 198.079,A -85,B 0,C 180,E1 -2180.078,E2 -2180.078} C_VEL
LIN {X 0,Y 573.197,Z 198.082,A -85,B 0,C 180,E1 -2182.339,E2 -2182.339} C_VEL
LIN {X 0,Y 573.207,Z 198.078,A -85,B 0,C 180,E1 -2185.412,E2 -2185.412} C_VEL
LIN {X 0,Y 573.2,Z 198.089,A -85,B 0,C 180,E1 -2188.567,E2 -2188.567} C_VEL
LIN {X 0,Y 573.191,Z 198.084,A -85,B 0,C 180,E1 -2190.996,E2 -2190.996} C_VEL
LIN {X 0,Y 573.214,Z 198.077,A -85,B 0,C 180,E1 -2193.523,E2 -2193.523} C_VEL
LIN {X 0,Y 573.188,Z 198.085,A -85,B 0,C 180,E1 -2196.054,E2 -2196.054} C_VEL
LIN {X 0,Y 573.214,Z 198.081,A -85,B 0,C 180,E1 -2198.704,E2 -2198.704} C_VEL
LIN {X 0,Y 573.221,Z 198.078,A -85,B 0,C 180,E1 -2201.596,E2 -2201.596} C_VEL
LIN {X 0,Y 573.209,Z 198.087,A -85,B 0,C 180,E1 -2204.336,E2 -2204.336} C_VEL
LIN {X 0,Y 573.216,Z 198.077,A -85,B 0,C 180,E1 -2207.361,E2 -2207.361} C_VEL
LIN {X 0,Y 573.224,Z 198.082,A -85,B 0,C 180,E1 -2210.394,E2 -2210.394} C_VEL
LIN {X 0,Y 573.241,Z 198.075,A -85,B 0,C 180,E1 -2213.079,E2 -2213.079} C_VEL
LIN {X 0,Y 573.255,Z 198.077,A -85,B 0,C 180,E1 -2215.673,E2 -2215.673} C_VEL
LIN {X 0,Y 573.23,Z 198.083,A -85,B 0,C 180,E1 -2218.186,E2 -2218.186} C_VEL
LIN {X 0,Y 573.255,Z 198.074,A -85,B 0,C 180,E1 -2220.635,E2 -2220.635} C_VEL
LIN {X 0,Y 573.251,Z 198.082,A -85,B 0,C 180,E1 -2223.811,E2 -2223.811} C_VEL
LIN {X 0,Y 573.269,Z 198.209,A -85,B 0,C 180,E1 -2226.159,E2 -2226.159} C_VEL
LIN {X 0,Y 574.003,Z 203.552,A -85,B 0,C 180,E1 -2226.934,E2 -2226.934} C_VEL
LIN {X 0,Y 573.853,Z 223.978,A -85,B 0,C 180,E1 -2229.759,E2 -2229.759} C_VEL
LIN {X 0,Y 573.615,Z 245.479,A -85,B 0,C 180,E1 -2232.735,E2 -2232.735} C_VEL
LIN {X 0,Y 573.464,Z 264.929,A -85,B 0,C 180,E1 -2235.401,E2 -2235.401} C_VEL
LIN {X 0,Y 573.417,Z 270.522,A -85,B 0,C 180,E1 -2236.161,E2 -2236.161} C_VEL
LIN {X 0,Y 574.063,Z 276.509,A -85,B 0,C 180,E1 -2236.256,E2 -2236.256} C_VEL
LIN {X 0,Y 573.879,Z 378.94,A -85,B 0,C 180,E1 -2237.557,E2 -2237.557} C_VEL
LIN {X 0,Y 573.798,Z 392.213,A -85,B 0,C 180,E1 -2237.87,E2 -2237.87} C_VEL
LIN {X 0,Y 573.702,Z 404.371,A -85,B 0,C 180,E1 -2238.294,E2 -2238.294} C_VEL
LIN {X 0,Y 573.58,Z 416.622,A -85,B 0,C 180,E1 -2238.873,E2 -2238.873} C_VEL
LIN {X 0,Y 573.436,Z 428.195,A -85,B 0,C 180,E1 -2239.585,E2 -2239.585} C_VEL
LIN {X 0,Y 573.332,Z 438.597,A -85,B 0,C 180,E1 -2240.385,E2 -2240.385} C_VEL
LIN {X 0,Y 573.241,Z 447.108,A -85,B 0,C 180,E1 -2241.184,E2 -2241.184} C_VEL
LIN {X 0,Y 573.161,Z 454.956,A -85,B 0,C 180,E1 -2242.07,E2 -2242.07} C_VEL
LIN {X 0,Y 573.074,Z 462.578,A -85,B 0,C 180,E1 -2243.126,E2 -2243.126} C_VEL
LIN {X 0,Y 573.07,Z 469.676,A -85,B 0,C 180,E1 -2244.369,E2 -2244.369} C_VEL
LIN {X 0,Y 573.029,Z 474.369,A -85,B 0,C 180,E1 -2245.427,E2 -2245.427} C_VEL
LIN {X 0,Y 573.022,Z 477.955,A -85,B 0,C 180,E1 -2246.483,E2 -2246.483} C_VEL
LIN {X 0,Y 572.959,Z 479.806,A -85,B 0,C 180,E1 -2247.187,E2 -2247.187} C_VEL
LIN {X 0,Y 572.94,Z 481.196,A -85,B 0,C 180,E1 -2247.89,E2 -2247.89} C_VEL
